LIN {X 0,Y 266.686,Z 225.636,A -85,B 0,C 180,E1 -19024.514,E2 -19024.514} C_VEL
LIN {X 0,Y 268.475,Z 213.294,A -85,B 0,C 180,E1 -19025.614,E2 -19025.614} C_VEL
LIN {X 0,Y 269.905,Z 200.622,A -85,B 0,C 180,E1 -19026.396,E2 -19026.396} C_VEL
LIN {X 0,Y 270.797,Z 187.768,A -85,B 0,C 180,E1 -19026.906,E2 -19026.906} C_VEL
LIN {X 0,Y 272.877,Z 131.801,A -85,B 0,C 180,E1 -19028.371,E2 -19028.371} C_VEL
LIN {X 0,Y 266.197,Z 116.896,A -85,B 0,C 180,E1 -19029.859,E2 -19029.859} C_VEL
LIN {X 0,Y 258.675,Z 102.48,A -85,B 0,C 180,E1 -19031.584,E2 -19031.584} C_VEL
LIN {X 0,Y 252.881,Z 93.623,A -85,B 0,C 180,E1 -19032.932,E2 -19032.932} C_VEL
LIN {X 0,Y 251.097,Z 90.671,A -85,B 0,C 180,E1 -19033.374,E2 -19033.374} C_VEL
LIN {X 0,Y 249.511,Z 88.379,A -85,B 0,C 180,E1 -19033.762,E2 -19033.762} C_VEL
LIN {X 0,Y 248.965,Z 86.456,A -85,B 0,C 180,E1 -19033.98,E2 -19033.98} C_VEL
LIN {X 0,Y 248.982,Z 86.472,A -85,B 0,C 180,E1 -19037.355,E2 -19037.355} C_VEL
LIN {X 0,Y 249.046,Z 86.459,A -85,B 0,C 180,E1 -19042.2,E2 -19042.2} C_VEL
LIN {X 0,Y 249.046,Z 86.459,A -85,B 0,C 180,E1 -19045.639,E2 -19045.639} C_VEL
LIN {X 0,Y 248.998,Z 86.463,A -85,B 0,C 180,E1 -19049.465,E2 -19049.465} C_VEL
LIN {X 0,Y 249.033,Z 86.454,A -85,B 0,C 180,E1 -19053.157,E2 -19053.157} C_VEL
LIN {X 0,Y 249.057,Z 86.45,A -85,B 0,C 180,E1 -19056.73,E2 -19056.73} C_VEL
LIN {X 0,Y 249.094,Z 86.457,A -85,B 0,C 180,E1 -19060.21,E2 -19060.21} C_VEL
LIN {X 0,Y 249.199,Z 86.435,A -85,B 0,C 180,E1 -19063.619,E2 -19063.619} C_VEL
LIN {X 0,Y 249.234,Z 86.424,A -85,B 0,C 180,E1 -19068.615,E2 -19068.615} C_VEL
LIN {X 0,Y 249.42,Z 86.413,A -85,B 0,C 180,E1 -19071.9,E2 -19071.9} C_VEL
LIN {X 0,Y 249.27,Z 86.425,A -85,B 0,C 180,E1 -19075.148,E2 -19075.148} C_VEL
LIN {X 0,Y 249.648,Z 86.375,A -85,B 0,C 180,E1 -19078.702,E2 -19078.702} C_VEL
LIN {X 0,Y 249.289,Z 86.416,A -85,B 0,C 180,E1 -19079.602,E2 -19079.602} C_VEL
LIN {X 0,Y 247.208,Z 86.686,A -85,B 0,C 180,E1 -19081.364,E2 -19081.364} C_VEL
LIN {X 0,Y 243.334,Z 87.169,A -85,B 0,C 180,E1 -19084.017,E2 -19084.017} C_VEL
LIN {X 0,Y 242.334,Z 87.282,A -85,B 0,C 180,E1 -19085.405,E2 -19085.405} C_VEL
LIN {X 0,Y 242.295,Z 87.285,A -85,B 0,C 180,E1 -19085.876,E2 -19085.876} C_VEL
LIN {X 0,Y 242.333,Z 87.296,A -85,B 0,C 180,E1 -19089.578,E2 -19089.578} C_VEL
LIN {X 0,Y 242.142,Z 87.321,A -85,B 0,C 180,E1 -19095.142,E2 -19095.142} C_VEL
LIN {X 0,Y 242.063,Z 87.326,A -85,B 0,C 180,E1 -19098.625,E2 -19098.625} C_VEL
LIN {X 0,Y 242.016,Z 87.324,A -85,B 0,C 180,E1 -19102.179,E2 -19102.179} C_VEL
LIN {X 0,Y 242.069,Z 87.326,A -85,B 0,C 180,E1 -19105.838,E2 -19105.838} C_VEL
LIN {X 0,Y 242.033,Z 87.335,A -85,B 0,C 180,E1 -19109.58,E2 -19109.58} C_VEL
LIN {X 0,Y 241.983,Z 87.341,A -85,B 0,C 180,E1 -19113.492,E2 -19113.492} C_VEL
LIN {X 0,Y 241.989,Z 87.313,A -85,B 0,C 180,E1 -19117.582,E2 -19117.582} C_VEL
LIN {X 0,Y 241.939,Z 87.346,A -85,B 0,C 180,E1 -19121.922,E2 -19121.922} C_VEL
LIN {X 0,Y 241.987,Z 87.448,A -85,B 0,C 180,E1 -19125.281,E2 -19125.281} C_VEL
LIN {X 0,Y 244.136,Z 95.03,A -85,B 0,C 180,E1 -19129.083,E2 -19129.083} C_VEL
LIN {X 0,Y 246.23,Z 102.697,A -85,B 0,C 180,E1 -19132.554,E2 -19132.554} C_VEL
LIN {X 0,Y 248.552,Z 107.076,A -85,B 0,C 180,E1 -19133.167,E2 -19133.167} C_VEL
LIN {X 0,Y 255.724,Z 121.344,A -85,B 0,C 180,E1 -19134.984,E2 -19134.984} C_VEL
LIN {X 0,Y 261.909,Z 135.149,A -85,B 0,C 180,E1 -19136.488,E2 -19136.488} C_VEL
LIN {X 0,Y 265.889,Z 160.561,A -85,B 0,C 180,E1 -19137.938,E2 -19137.938} C_VEL
LIN {X 0,Y 263.797,Z 212.777,A -85,B 0,C 180,E1 -19139.366,E2 -19139.366} C_VEL
LIN {X 0,Y 262.461,Z 226.52,A -85,B 0,C 180,E1 -19140.028,E2 -19140.028} C_VEL
LIN {X 0,Y 260.406,Z 239.381,A -85,B 0,C 180,E1 -19140.935,E2 -19140.935} C_VEL
LIN {X 0,Y 257.946,Z 251.892,A -85,B 0,C 180,E1 -19142.186,E2 -19142.186} C_VEL
LIN {X 0,Y 255.344,Z 263.061,A -85,B 0,C 180,E1 -19143.652,E2 -19143.652} C_VEL
LIN {X 0,Y 252.648,Z 273.135,A -85,B 0,C 180,E1 -19145.338,E2 -19145.338} C_VEL
LIN {X 0,Y 249.903,Z 282.245,A -85,B 0,C 180,E1 -19147.251,E2 -19147.251} C_VEL
LIN {X 0,Y 247.152,Z 291.145,A -85,B 0,C 180,E1 -19149.614,E2 -19149.614} C_VEL
LIN {X 0,Y 244.923,Z 298.327,A -85,B 0,C 180,E1 -19152.032,E2 -19152.032} C_VEL
LIN {X 0,Y 243.352,Z 303.192,A -85,B 0,C 180,E1 -19154.076,E2 -19154.076} C_VEL
LIN {X 0,Y 241.72,Z 307.936,A -85,B 0,C 180,E1 -19156.549,E2 -19156.549} C_VEL
LIN {X 0,Y 240.769,Z 311.589,A -85,B 0,C 180,E1 -19159.062,E2 -19159.062} C_VEL
LIN {X 0,Y 240.145,Z 314.246,A -85,B 0,C 180,E1 -19161.585,E2 -19161.585} C_VEL
LIN {X 0,Y 239.898,Z 315.513,A -85,B 0,C 180,E1 -19163.27,E2 -19163.27} C_VEL
LIN {X 0,Y 239.845,Z 316.4,A -85,B 0,C 180,E1 -19165.053,E2 -19165.053} C_VEL
LIN {X 0,Y 239.971,Z 316.852,A -85,B 0,C 180,E1 -19168.321,E2 -19168.321} C_VEL
LIN {X 0,Y 240.02,Z 316.509,A -85,B 0,C 180,E1 -19169.999,E2 -19169.999} C_VEL
LIN {X 0,Y 239.992,Z 315.759,A -85,B 0,C 180,E1 -19171.678,E2 -19171.678} C_VEL
LIN {X 0,Y 239.93,Z 314.556,A -85,B 0,C 180,E1 -19173.358,E2 -19173.358} C_VEL
LIN {X 0,Y 239.889,Z 311.975,A -85,B 0,C 180,E1 -19175.885,E2 -19175.885} C_VEL
LIN {X 0,Y 240.128,Z 308.368,A -85,B 0,C 180,E1 -19178.414,E2 -19178.414} C_VEL
LIN {X 0,Y 240.607,Z 303.629,A -85,B 0,C 180,E1 -19180.944,E2 -19180.944} C_VEL
LIN {X 0,Y 241.486,Z 297.624,A -85,B 0,C 180,E1 -19183.463,E2 -19183.463} C_VEL
LIN {X 0,Y 242.785,Z 290.138,A -85,B 0,C 180,E1 -19185.962,E2 -19185.962} C_VEL
LIN {X 0,Y 244.271,Z 282.197,A -85,B 0,C 180,E1 -19188.098,E2 -19188.098} C_VEL
LIN {X 0,Y 245.678,Z 273.231,A -85,B 0,C 180,E1 -19190.076,E2 -19190.076} C_VEL
LIN {X 0,Y 247.634,Z 262.952,A -85,B 0,C 180,E1 -19191.869,E2 -19191.869} C_VEL
LIN {X 0,Y 249.5,Z 251.528,A -85,B 0,C 180,E1 -19193.445,E2 -19193.445} C_VEL
LIN {X 0,Y 251.171,Z 239.655,A -85,B 0,C 180,E1 -19194.706,E2 -19194.706} C_VEL
LIN {X 0,Y 252.699,Z 226.572,A -85,B 0,C 180,E1 -19195.701,E2 -19195.701} C_VEL
LIN {X 0,Y 253.626,Z 213.267,A -85,B 0,C 180,E1 -19196.389,E2 -19196.389} C_VEL
LIN {X 0,Y 255.41,Z 156.007,A -85,B 0,C 180,E1 -19197.998,E2 -19197.998} C_VEL
LIN {X 0,Y 251.667,Z 125.16,A -85,B 0,C 180,E1 -19199.347,E2 -19199.347} C_VEL
LIN {X 0,Y 250.229,Z 115.793,A -85,B 0,C 180,E1 -19199.802,E2 -19199.802} C_VEL
LIN {X 0,Y 245.606,Z 103.483,A -85,B 0,C 180,E1 -19200.789,E2 -19200.789} C_VEL
LIN {X 0,Y 243.41,Z 93.051,A -85,B 0,C 180,E1 -19204.766,E2 -19204.766} C_VEL
LIN {X 0,Y 242.051,Z 87.339,A -85,B 0,C 180,E1 -19207.09,E2 -19207.09} C_VEL
LIN {X 0,Y 241.942,Z 87.348,A -85,B 0,C 180,E1 -19211.921,E2 -19211.921} C_VEL
LIN {X 0,Y 241.926,Z 87.349,A -85,B 0,C 180,E1 -19216.573,E2 -19216.573} C_VEL
LIN {X 0,Y 241.955,Z 87.332,A -85,B 0,C 180,E1 -19220.281,E2 -19220.281} C_VEL
LIN {X 0,Y 241.986,Z 87.339,A -85,B 0,C 180,E1 -19224.489,E2 -19224.489} C_VEL
LIN {X 0,Y 241.974,Z 87.343,A -85,B 0,C 180,E1 -19228.48,E2 -19228.48} C_VEL
LIN {X 0,Y 242.008,Z 87.336,A -85,B 0,C 180,E1 -19232.313,E2 -19232.313} C_VEL
LIN {X 0,Y 242.057,Z 87.332,A -85,B 0,C 180,E1 -19236.016,E2 -19236.016} C_VEL
LIN {X 0,Y 242.036,Z 87.324,A -85,B 0,C 180,E1 -19239.608,E2 -19239.608} C_VEL
LIN {X 0,Y 242.162,Z 87.319,A -85,B 0,C 180,E1 -19243.278,E2 -19243.278} C_VEL
LIN {X 0,Y 242.18,Z 87.305,A -85,B 0,C 180,E1 -19248.28,E2 -19248.28} C_VEL
LIN {X 0,Y 242.4,Z 87.289,A -85,B 0,C 180,E1 -19251.665,E2 -19251.665} C_VEL
LIN {X 0,Y 242.422,Z 87.285,A -85,B 0,C 180,E1 -19253.341,E2 -19253.341} C_VEL
LIN {X 0,Y 242.634,Z 87.258,A -85,B 0,C 180,E1 -19258.341,E2 -19258.341} C_VEL
LIN {X 0,Y 242.633,Z 87.261,A -85,B 0,C 180,E1 -19261.66,E2 -19261.66} C_VEL
LIN {X 0,Y 242.408,Z 87.284,A -85,B 0,C 180,E1 -19266.66,E2 -19266.66} C_VEL
LIN {X 0,Y 242.266,Z 87.304,A -85,B 0,C 180,E1 -19270.024,E2 -19270.024} C_VEL
LIN {X 0,Y 242.167,Z 87.312,A -85,B 0,C 180,E1 -19275.141,E2 -19275.141} C_VEL
LIN {X 0,Y 242.073,Z 87.327,A -85,B 0,C 180,E1 -19278.625,E2 -19278.625} C_VEL
LIN {X 0,Y 242.013,Z 87.329,A -85,B 0,C 180,E1 -19282.18,E2 -19282.18} C_VEL
LIN {X 0,Y 242.067,Z 87.33,A -85,B 0,C 180,E1 -19285.839,E2 -19285.839} C_VEL
LIN {X 0,Y 242.007,Z 87.338,A -85,B 0,C 180,E1 -19289.584,E2 -19289.584} C_VEL
LIN {X 0,Y 241.981,Z 87.342,A -85,B 0,C 180,E1 -19293.493,E2 -19293.493} C_VEL
LIN {X 0,Y 241.985,Z 87.34,A -85,B 0,C 180,E1 -19297.583,E2 -19297.583} C_VEL
LIN {X 0,Y 241.912,Z 87.349,A -85,B 0,C 180,E1 -19301.928,E2 -19301.928} C_VEL
LIN {X 0,Y 241.925,Z 87.351,A -85,B 0,C 180,E1 -19306.574,E2 -19306.574} C_VEL
LIN {X 0,Y 241.996,Z 87.34,A -85,B 0,C 180,E1 -19311.641,E2 -19311.641} C_VEL
LIN {X 0,Y 241.981,Z 87.343,A -85,B 0,C 180,E1 -19314.489,E2 -19314.489} C_VEL
LIN {X 0,Y 241.955,Z 87.346,A -85,B 0,C 180,E1 -19318.478,E2 -19318.478} C_VEL
LIN {X 0,Y 241.966,Z 87.336,A -85,B 0,C 180,E1 -19322.308,E2 -19322.308} C_VEL
LIN {X 0,Y 242.031,Z 87.516,A -85,B 0,C 180,E1 -19325.996,E2 -19325.996} C_VEL
LIN {X 0,Y 243.188,Z 90.492,A -85,B 0,C 180,E1 -19326.241,E2 -19326.241} C_VEL
LIN {X 0,Y 250.953,Z 106.159,A -85,B 0,C 180,E1 -19327.677,E2 -19327.677} C_VEL
LIN {X 0,Y 256.395,Z 121.2,A -85,B 0,C 180,E1 -19328.745,E2 -19328.745} C_VEL
LIN {X 0,Y 254.142,Z 192.259,A -85,B 0,C 180,E1 -19330.725,E2 -19330.725} C_VEL
LIN {X 0,Y 253.29,Z 205.938,A -85,B 0,C 180,E1 -19331.445,E2 -19331.445} C_VEL
LIN {X 0,Y 252.18,Z 218.733,A -85,B 0,C 180,E1 -19332.463,E2 -19332.463} C_VEL
LIN {X 0,Y 250.796,Z 230.411,A -85,B 0,C 180,E1 -19333.727,E2 -19333.727} C_VEL
LIN {X 0,Y 249.149,Z 241.669,A -85,B 0,C 180,E1 -19335.294,E2 -19335.294} C_VEL
LIN {X 0,Y 247.422,Z 251.831,A -85,B 0,C 180,E1 -19337.075,E2 -19337.075} C_VEL
LIN {X 0,Y 245.507,Z 261.778,A -85,B 0,C 180,E1 -19339.277,E2 -19339.277} C_VEL
LIN {X 0,Y 243.847,Z 270.522,A -85,B 0,C 180,E1 -19341.715,E2 -19341.715} C_VEL
LIN {X 0,Y 242.477,Z 277.536,A -85,B 0,C 180,E1 -19344.178,E2 -19344.178} C_VEL
LIN {X 0,Y 241.47,Z 283.133,A -85,B 0,C 180,E1 -19346.663,E2 -19346.663} C_VEL
LIN {X 0,Y 240.784,Z 287.545,A -85,B 0,C 180,E1 -19349.164,E2 -19349.164} C_VEL
LIN {X 0,Y 240.255,Z 290.905,A -85,B 0,C 180,E1 -19351.677,E2 -19351.677} C_VEL
LIN {X 0,Y 240.145,Z 292.572,A -85,B 0,C 180,E1 -19353.356,E2 -19353.356} C_VEL
LIN {X 0,Y 240.099,Z 294.188,A -85,B 0,C 180,E1 -19355.596,E2 -19355.596} C_VEL
LIN {X 0,Y 239.998,Z 295.194,A -85,B 0,C 180,E1 -19358.42,E2 -19358.42} C_VEL
LIN {X 0,Y 240.264,Z 294.941,A -85,B 0,C 180,E1 -19361.816,E2 -19361.816} C_VEL
LIN {X 0,Y 240.673,Z 294.231,A -85,B 0,C 180,E1 -19363.51,E2 -19363.51} C_VEL
LIN {X 0,Y 241.59,Z 292.169,A -85,B 0,C 180,E1 -19366.26,E2 -19366.26} C_VEL
LIN {X 0,Y 243.041,Z 288.332,A -85,B 0,C 180,E1 -19369.424,E2 -19369.424} C_VEL
LIN {X 0,Y 244.642,Z 284.067,A -85,B 0,C 180,E1 -19371.93,E2 -19371.93} C_VEL
LIN {X 0,Y 246.56,Z 278.599,A -85,B 0,C 180,E1 -19374.408,E2 -19374.408} C_VEL
LIN {X 0,Y 248.962,Z 271.704,A -85,B 0,C 180,E1 -19376.851,E2 -19376.851} C_VEL
LIN {X 0,Y 251.23,Z 264.642,A -85,B 0,C 180,E1 -19378.853,E2 -19378.853} C_VEL
LIN {X 0,Y 253.991,Z 254.913,A -85,B 0,C 180,E1 -19381.064,E2 -19381.064} C_VEL
LIN {X 0,Y 256.369,Z 245.433,A -85,B 0,C 180,E1 -19382.781,E2 -19382.781} C_VEL
LIN {X 0,Y 258.848,Z 234.847,A -85,B 0,C 180,E1 -19384.291,E2 -19384.291} C_VEL
LIN {X 0,Y 261.136,Z 223.08,A -85,B 0,C 180,E1 -19385.592,E2 -19385.592} C_VEL
LIN {X 0,Y 262.821,Z 210.853,A -85,B 0,C 180,E1 -19386.62,E2 -19386.62} C_VEL
LIN {X 0,Y 264.272,Z 197.71,A -85,B 0,C 180,E1 -19387.375,E2 -19387.375} C_VEL
LIN {X 0,Y 265.023,Z 184.983,A -85,B 0,C 180,E1 -19387.828,E2 -19387.828} C_VEL
LIN {X 0,Y 267.04,Z 133.98,A -85,B 0,C 180,E1 -19389.171,E2 -19389.171} C_VEL
LIN {X 0,Y 261.154,Z 120.766,A -85,B 0,C 180,E1 -19390.542,E2 -19390.542} C_VEL
LIN {X 0,Y 253.955,Z 106.895,A -85,B 0,C 180,E1 -19392.261,E2 -19392.261} C_VEL
LIN {X 0,Y 246.423,Z 95.208,A -85,B 0,C 180,E1 -19394.113,E2 -19394.113} C_VEL
LIN {X 0,Y 244.287,Z 91.787,A -85,B 0,C 180,E1 -19394.673,E2 -19394.673} C_VEL
LIN {X 0,Y 242.546,Z 89.488,A -85,B 0,C 180,E1 -19395.122,E2 -19395.122} C_VEL
LIN {X 0,Y 241.914,Z 87.332,A -85,B 0,C 180,E1 -19395.373,E2 -19395.373} C_VEL
LIN {X 0,Y 241.907,Z 87.348,A -85,B 0,C 180,E1 -19399.058,E2 -19399.058} C_VEL
LIN {X 0,Y 241.987,Z 87.34,A -85,B 0,C 180,E1 -19402.417,E2 -19402.417} C_VEL
LIN {X 0,Y 241.982,Z 87.343,A -85,B 0,C 180,E1 -19406.507,E2 -19406.507} C_VEL
LIN {X 0,Y 241.975,Z 87.344,A -85,B 0,C 180,E1 -19410.615,E2 -19410.615} C_VEL
LIN {X 0,Y 242.036,Z 87.334,A -85,B 0,C 180,E1 -19414.179,E2 -19414.179} C_VEL
LIN {X 0,Y 242.025,Z 87.329,A -85,B 0,C 180,E1 -19418.316,E2 -19418.316} C_VEL
LIN {X 0,Y 242.131,Z 87.312,A -85,B 0,C 180,E1 -19423.306,E2 -19423.306} C_VEL
LIN {X 0,Y 242.169,Z 87.302,A -85,B 0,C 180,E1 -19428.278,E2 -19428.278} C_VEL
LIN {X 0,Y 242.374,Z 87.293,A -85,B 0,C 180,E1 -19431.663,E2 -19431.663} C_VEL
LIN {X 0,Y 242.4,Z 87.274,A -85,B 0,C 180,E1 -19433.34,E2 -19433.34} C_VEL
LIN {X 0,Y 242.608,Z 87.252,A -85,B 0,C 180,E1 -19438.692,E2 -19438.692} C_VEL
LIN {X 0,Y 242.623,Z 87.257,A -85,B 0,C 180,E1 -19441.66,E2 -19441.66} C_VEL
LIN {X 0,Y 242.295,Z 87.285,A -85,B 0,C 180,E1 -19445.876,E2 -19445.876} C_VEL
LIN {X 0,Y 241.711,Z 87.366,A -85,B 0,C 180,E1 -19447.263,E2 -19447.263} C_VEL
LIN {X 0,Y 240.11,Z 87.574,A -85,B 0,C 180,E1 -19448.624,E2 -19448.624} C_VEL
LIN {X 0,Y 236.236,Z 88.046,A -85,B 0,C 180,E1 -19451.363,E2 -19451.363} C_VEL
LIN {X 0,Y 235.147,Z 88.18,A -85,B 0,C 180,E1 -19452.796,E2 -19452.796} C_VEL
LIN {X 0,Y 235.066,Z 88.192,A -85,B 0,C 180,E1 -19453.283,E2 -19453.283} C_VEL
LIN {X 0,Y 235.052,Z 88.189,A -85,B 0,C 180,E1 -19457.397,E2 -19457.397} C_VEL
LIN {X 0,Y 234.996,Z 88.198,A -85,B 0,C 180,E1 -19462.009,E2 -19462.009} C_VEL
LIN {X 0,Y 234.972,Z 88.205,A -85,B 0,C 180,E1 -19466.657,E2 -19466.657} C_VEL
LIN {X 0,Y 234.934,Z 88.212,A -85,B 0,C 180,E1 -19470.567,E2 -19470.567} C_VEL
LIN {X 0,Y 234.929,Z 88.201,A -85,B 0,C 180,E1 -19474.638,E2 -19474.638} C_VEL
LIN {X 0,Y 234.944,Z 88.212,A -85,B 0,C 180,E1 -19478.944,E2 -19478.944} C_VEL
LIN {X 0,Y 234.896,Z 88.281,A -85,B 0,C 180,E1 -19483.96,E2 -19483.96} C_VEL
LIN {X 0,Y 237.023,Z 95.585,A -85,B 0,C 180,E1 -19487.84,E2 -19487.84} C_VEL
LIN {X 0,Y 238.883,Z 102.23,A -85,B 0,C 180,E1 -19491.026,E2 -19491.026} C_VEL
LIN {X 0,Y 241.091,Z 106.391,A -85,B 0,C 180,E1 -19491.655,E2 -19491.655} C_VEL
LIN {X 0,Y 246.988,Z 117.484,A -85,B 0,C 180,E1 -19493.252,E2 -19493.252} C_VEL
LIN {X 0,Y 253.517,Z 131.294,A -85,B 0,C 180,E1 -19494.948,E2 -19494.948} C_VEL
LIN {X 0,Y 256.548,Z 138.573,A -85,B 0,C 180,E1 -19495.722,E2 -19495.722} C_VEL
LIN {X 0,Y 260.07,Z 161.624,A -85,B 0,C 180,E1 -19497.078,E2 -19497.078} C_VEL
LIN {X 0,Y 257.937,Z 212.151,A -85,B 0,C 180,E1 -19498.478,E2 -19498.478} C_VEL
LIN {X 0,Y 256.643,Z 225.227,A -85,B 0,C 180,E1 -19499.105,E2 -19499.105} C_VEL
LIN {X 0,Y 254.648,Z 237.853,A -85,B 0,C 180,E1 -19499.984,E2 -19499.984} C_VEL
LIN {X 0,Y 252.439,Z 249.089,A -85,B 0,C 180,E1 -19501.07,E2 -19501.07} C_VEL
LIN {X 0,Y 249.994,Z 259.425,A -85,B 0,C 180,E1 -19502.363,E2 -19502.363} C_VEL
LIN {X 0,Y 247.104,Z 270.114,A -85,B 0,C 180,E1 -19504.068,E2 -19504.068} C_VEL
LIN {X 0,Y 243.883,Z 280.635,A -85,B 0,C 180,E1 -19506.206,E2 -19506.206} C_VEL
LIN {X 0,Y 240.926,Z 289.756,A -85,B 0,C 180,E1 -19508.614,E2 -19508.614} C_VEL
LIN {X 0,Y 238.574,Z 297.128,A -85,B 0,C 180,E1 -19511.092,E2 -19511.092} C_VEL
LIN {X 0,Y 236.518,Z 303.063,A -85,B 0,C 180,E1 -19513.603,E2 -19513.603} C_VEL
LIN {X 0,Y 234.793,Z 307.765,A -85,B 0,C 180,E1 -19516.145,E2 -19516.145} C_VEL
LIN {X 0,Y 233.766,Z 311.379,A -85,B 0,C 180,E1 -19518.73,E2 -19518.73} C_VEL
LIN {X 0,Y 233.093,Z 314,A -85,B 0,C 180,E1 -19521.329,E2 -19521.329} C_VEL
LIN {X 0,Y 232.819,Z 315.249,A -85,B 0,C 180,E1 -19523.064,E2 -19523.064} C_VEL
LIN {X 0,Y 232.745,Z 316.188,A -85,B 0,C 180,E1 -19525.185,E2 -19525.185} C_VEL
LIN {X 0,Y 232.898,Z 316.524,A -85,B 0,C 180,E1 -19528.27,E2 -19528.27} C_VEL
LIN {X 0,Y 232.947,Z 316.165,A -85,B 0,C 180,E1 -19529.999,E2 -19529.999} C_VEL
LIN {X 0,Y 232.92,Z 315.383,A -85,B 0,C 180,E1 -19531.729,E2 -19531.729} C_VEL
LIN {X 0,Y 232.801,Z 312.753,A -85,B 0,C 180,E1 -19534.974,E2 -19534.974} C_VEL
LIN {X 0,Y 232.966,Z 309.225,A -85,B 0,C 180,E1 -19537.802,E2 -19537.802} C_VEL
LIN {X 0,Y 233.391,Z 304.837,A -85,B 0,C 180,E1 -19540.409,E2 -19540.409} C_VEL
LIN {X 0,Y 234.155,Z 299.239,A -85,B 0,C 180,E1 -19543.009,E2 -19543.009} C_VEL
LIN {X 0,Y 235.443,Z 292.254,A -85,B 0,C 180,E1 -19545.583,E2 -19545.583} C_VEL
LIN {X 0,Y 237.033,Z 284.158,A -85,B 0,C 180,E1 -19547.957,E2 -19547.957} C_VEL
LIN {X 0,Y 238.594,Z 274.467,A -85,B 0,C 180,E1 -19550.249,E2 -19550.249} C_VEL
LIN {X 0,Y 240.547,Z 264.596,A -85,B 0,C 180,E1 -19552.096,E2 -19552.096} C_VEL
LIN {X 0,Y 242.469,Z 253.719,A -85,B 0,C 180,E1 -19553.713,E2 -19553.713} C_VEL
LIN {X 0,Y 244.299,Z 241.486,A -85,B 0,C 180,E1 -19555.108,E2 -19555.108} C_VEL
LIN {X 0,Y 245.939,Z 228.696,A -85,B 0,C 180,E1 -19556.176,E2 -19556.176} C_VEL
LIN {X 0,Y 246.944,Z 215.883,A -85,B 0,C 180,E1 -19556.916,E2 -19556.916} C_VEL
LIN {X 0,Y 247.636,Z 199.657,A -85,B 0,C 180,E1 -19557.457,E2 -19557.457} C_VEL
LIN {X 0,Y 248.905,Z 156.447,A -85,B 0,C 180,E1 -19558.673,E2 -19558.673} C_VEL
LIN {X 0,Y 245.449,Z 127.202,A -85,B 0,C 180,E1 -19559.991,E2 -19559.991} C_VEL
LIN {X 0,Y 244.025,Z 118.013,A -85,B 0,C 180,E1 -19560.456,E2 -19560.456} C_VEL
LIN {X 0,Y 239.176,Z 105.676,A -85,B 0,C 180,E1 -19561.463,E2 -19561.463} C_VEL
LIN {X 0,Y 238.303,Z 103.126,A -85,B 0,C 180,E1 -19561.713,E2 -19561.713} C_VEL
LIN {X 0,Y 236.632,Z 95.125,A -85,B 0,C 180,E1 -19564.87,E2 -19564.87} C_VEL
LIN {X 0,Y 234.976,Z 88.221,A -85,B 0,C 180,E1 -19567.817,E2 -19567.817} C_VEL
LIN {X 0,Y 234.891,Z 88.226,A -85,B 0,C 180,E1 -19571.582,E2 -19571.582} C_VEL
LIN {X 0,Y 234.887,Z 88.227,A -85,B 0,C 180,E1 -19575.897,E2 -19575.897} C_VEL
LIN {X 0,Y 234.881,Z 88.225,A -85,B 0,C 180,E1 -19578.832,E2 -19578.832} C_VEL
LIN {X 0,Y 234.916,Z 88.203,A -85,B 0,C 180,E1 -19581.079,E2 -19581.079} C_VEL
LIN {X 0,Y 234.929,Z 88.222,A -85,B 0,C 180,E1 -19585.362,E2 -19585.362} C_VEL
LIN {X 0,Y 234.931,Z 88.221,A -85,B 0,C 180,E1 -19589.432,E2 -19589.432} C_VEL
LIN {X 0,Y 234.993,Z 88.206,A -85,B 0,C 180,E1 -19593.794,E2 -19593.794} C_VEL
LIN {X 0,Y 235.011,Z 88.201,A -85,B 0,C 180,E1 -19598.97,E2 -19598.97} C_VEL
LIN {X 0,Y 235.096,Z 88.2,A -85,B 0,C 180,E1 -19603.059,E2 -19603.059} C_VEL
LIN {X 0,Y 235.114,Z 88.183,A -85,B 0,C 180,E1 -19607.922,E2 -19607.922} C_VEL
LIN {X 0,Y 235.331,Z 88.17,A -85,B 0,C 180,E1 -19611.413,E2 -19611.413} C_VEL
LIN {X 0,Y 235.373,Z 88.163,A -85,B 0,C 180,E1 -19613.141,E2 -19613.141} C_VEL
LIN {X 0,Y 235.593,Z 88.134,A -85,B 0,C 180,E1 -19618.291,E2 -19618.291} C_VEL
LIN {X 0,Y 235.593,Z 88.138,A -85,B 0,C 180,E1 -19621.71,E2 -19621.71} C_VEL
LIN {X 0,Y 235.359,Z 88.161,A -85,B 0,C 180,E1 -19626.86,E2 -19626.86} C_VEL
LIN {X 0,Y 235.212,Z 88.181,A -85,B 0,C 180,E1 -19630.328,E2 -19630.328} C_VEL
LIN {X 0,Y 235.114,Z 88.193,A -85,B 0,C 180,E1 -19635.607,E2 -19635.607} C_VEL
LIN {X 0,Y 235.009,Z 88.207,A -85,B 0,C 180,E1 -19639.206,E2 -19639.206} C_VEL
LIN {X 0,Y 234.961,Z 88.208,A -85,B 0,C 180,E1 -19642.883,E2 -19642.883} C_VEL
LIN {X 0,Y 234.968,Z 88.214,A -85,B 0,C 180,E1 -19646.658,E2 -19646.658} C_VEL
LIN {X 0,Y 234.923,Z 88.22,A -85,B 0,C 180,E1 -19650.57,E2 -19650.57} C_VEL
LIN {X 0,Y 234.927,Z 88.221,A -85,B 0,C 180,E1 -19654.639,E2 -19654.639} C_VEL
LIN {X 0,Y 234.912,Z 88.224,A -85,B 0,C 180,E1 -19658.936,E2 -19658.936} C_VEL
LIN {X 0,Y 234.865,Z 88.229,A -85,B 0,C 180,E1 -19663.492,E2 -19663.492} C_VEL
LIN {X 0,Y 234.878,Z 88.229,A -85,B 0,C 180,E1 -19666.513,E2 -19666.513} C_VEL
LIN {X 0,Y 234.919,Z 88.222,A -85,B 0,C 180,E1 -19671.079,E2 -19671.079} C_VEL
LIN {X 0,Y 234.927,Z 88.22,A -85,B 0,C 180,E1 -19675.362,E2 -19675.362} C_VEL
LIN {X 0,Y 234.901,Z 88.222,A -85,B 0,C 180,E1 -19679.428,E2 -19679.428} C_VEL
LIN {X 0,Y 234.966,Z 88.216,A -85,B 0,C 180,E1 -19684.394,E2 -19684.394} C_VEL
LIN {X 0,Y 234.994,Z 88.214,A -85,B 0,C 180,E1 -19685.069,E2 -19685.069} C_VEL
LIN {X 0,Y 236.009,Z 91.114,A -85,B 0,C 180,E1 -19685.329,E2 -19685.329} C_VEL
LIN {X 0,Y 244.946,Z 108.846,A -85,B 0,C 180,E1 -19687.056,E2 -19687.056} C_VEL
LIN {X 0,Y 249.986,Z 122.737,A -85,B 0,C 180,E1 -19688.088,E2 -19688.088} C_VEL
LIN {X 0,Y 247.68,Z 191.908,A -85,B 0,C 180,E1 -19690.047,E2 -19690.047} C_VEL
LIN {X 0,Y 246.882,Z 204.939,A -85,B 0,C 180,E1 -19690.729,E2 -19690.729} C_VEL
LIN {X 0,Y 245.681,Z 218.154,A -85,B 0,C 180,E1 -19691.768,E2 -19691.768} C_VEL
LIN {X 0,Y 244.278,Z 230.044,A -85,B 0,C 180,E1 -19693.065,E2 -19693.065} C_VEL
LIN {X 0,Y 242.541,Z 241.43,A -85,B 0,C 180,E1 -19694.669,E2 -19694.669} C_VEL
LIN {X 0,Y 240.757,Z 251.696,A -85,B 0,C 180,E1 -19696.496,E2 -19696.496} C_VEL
LIN {X 0,Y 238.931,Z 260.935,A -85,B 0,C 180,E1 -19698.549,E2 -19698.549} C_VEL
LIN {X 0,Y 237.116,Z 269.879,A -85,B 0,C 180,E1 -19701.048,E2 -19701.048} C_VEL
LIN {X 0,Y 235.671,Z 277.088,A -85,B 0,C 180,E1 -19703.58,E2 -19703.58} C_VEL
LIN {X 0,Y 234.691,Z 281.968,A -85,B 0,C 180,E1 -19705.707,E2 -19705.707} C_VEL
LIN {X 0,Y 233.917,Z 286.706,A -85,B 0,C 180,E1 -19708.279,E2 -19708.279} C_VEL
LIN {X 0,Y 233.284,Z 290.357,A -85,B 0,C 180,E1 -19710.864,E2 -19710.864} C_VEL
LIN {X 0,Y 233.051,Z 292.996,A -85,B 0,C 180,E1 -19713.458,E2 -19713.458} C_VEL
LIN {X 0,Y 233.032,Z 294.479,A -85,B 0,C 180,E1 -19715.582,E2 -19715.582} C_VEL
LIN {X 0,Y 232.906,Z 295.529,A -85,B 0,C 180,E1 -19718.678,E2 -19718.678} C_VEL
LIN {X 0,Y 233.237,Z 295.231,A -85,B 0,C 180,E1 -19722.177,E2 -19722.177} C_VEL
LIN {X 0,Y 233.704,Z 294.485,A -85,B 0,C 180,E1 -19723.921,E2 -19723.921} C_VEL
LIN {X 0,Y 234.613,Z 292.567,A -85,B 0,C 180,E1 -19726.545,E2 -19726.545} C_VEL
LIN {X 0,Y 235.78,Z 289.692,A -85,B 0,C 180,E1 -19729.141,E2 -19729.141} C_VEL
LIN {X 0,Y 237.351,Z 285.752,A -85,B 0,C 180,E1 -19731.724,E2 -19731.724} C_VEL
LIN {X 0,Y 239.484,Z 280.052,A -85,B 0,C 180,E1 -19734.529,E2 -19734.529} C_VEL
LIN {X 0,Y 242.11,Z 272.914,A -85,B 0,C 180,E1 -19737.207,E2 -19737.207} C_VEL
LIN {X 0,Y 244.946,Z 264.531,A -85,B 0,C 180,E1 -19739.666,E2 -19739.666} C_VEL
LIN {X 0,Y 247.715,Z 255.097,A -85,B 0,C 180,E1 -19741.84,E2 -19741.84} C_VEL
LIN {X 0,Y 250.042,Z 246.27,A -85,B 0,C 180,E1 -19743.478,E2 -19743.478} C_VEL
LIN {X 0,Y 252.607,Z 235.795,A -85,B 0,C 180,E1 -19745.018,E2 -19745.018} C_VEL
LIN {X 0,Y 254.989,Z 224.255,A -85,B 0,C 180,E1 -19746.341,E2 -19746.341} C_VEL
LIN {X 0,Y 256.643,Z 212.885,A -85,B 0,C 180,E1 -19747.352,E2 -19747.352} C_VEL
LIN {X 0,Y 258.232,Z 199.432,A -85,B 0,C 180,E1 -19748.172,E2 -19748.172} C_VEL
LIN {X 0,Y 259.127,Z 186.818,A -85,B 0,C 180,E1 -19748.653,E2 -19748.653} C_VEL
LIN {X 0,Y 261.218,Z 136.002,A -85,B 0,C 180,E1 -19750.019,E2 -19750.019} C_VEL
LIN {X 0,Y 255.346,Z 123.018,A -85,B 0,C 180,E1 -19751.447,E2 -19751.447} C_VEL
LIN {X 0,Y 249.181,Z 111.171,A -85,B 0,C 180,E1 -19752.987,E2 -19752.987} C_VEL
LIN {X 0,Y 241.952,Z 99.851,A -85,B 0,C 180,E1 -19754.844,E2 -19754.844} C_VEL
LIN {X 0,Y 239.574,Z 96.295,A -85,B 0,C 180,E1 -19755.484,E2 -19755.484} C_VEL
LIN {X 0,Y 237.264,Z 92.721,A -85,B 0,C 180,E1 -19756.131,E2 -19756.131} C_VEL
LIN {X 0,Y 235.438,Z 90.284,A -85,B 0,C 180,E1 -19756.64,E2 -19756.64} C_VEL
LIN {X 0,Y 234.873,Z 88.227,A -85,B 0,C 180,E1 -19756.902,E2 -19756.902} C_VEL
LIN {X 0,Y 234.921,Z 88.217,A -85,B 0,C 180,E1 -19761.078,E2 -19761.078} C_VEL
LIN {X 0,Y 234.926,Z 88.215,A -85,B 0,C 180,E1 -19765.36,E2 -19765.36} C_VEL
LIN {X 0,Y 234.898,Z 88.219,A -85,B 0,C 180,E1 -19769.427,E2 -19769.427} C_VEL
LIN {X 0,Y 234.971,Z 88.21,A -85,B 0,C 180,E1 -19773.807,E2 -19773.807} C_VEL
LIN {X 0,Y 234.994,Z 88.209,A -85,B 0,C 180,E1 -19778.968,E2 -19778.968} C_VEL
LIN {X 0,Y 235.067,Z 88.19,A -85,B 0,C 180,E1 -19783.085,E2 -19783.085} C_VEL
LIN {X 0,Y 235.101,Z 88.182,A -85,B 0,C 180,E1 -19787.921,E2 -19787.921} C_VEL
LIN {X 0,Y 235.314,Z 88.173,A -85,B 0,C 180,E1 -19791.411,E2 -19791.411} C_VEL
LIN {X 0,Y 235.351,Z 88.152,A -85,B 0,C 180,E1 -19793.139,E2 -19793.139} C_VEL
LIN {X 0,Y 235.581,Z 88.131,A -85,B 0,C 180,E1 -19798.29,E2 -19798.29} C_VEL
LIN {X 0,Y 235.582,Z 88.134,A -85,B 0,C 180,E1 -19801.709,E2 -19801.709} C_VEL
LIN {X 0,Y 235.356,Z 88.153,A -85,B 0,C 180,E1 -19806.86,E2 -19806.86} C_VEL
LIN {X 0,Y 235.215,Z 88.176,A -85,B 0,C 180,E1 -19810.327,E2 -19810.327} C_VEL
LIN {X 0,Y 235.066,Z 88.192,A -85,B 0,C 180,E1 -19813.283,E2 -19813.283} C_VEL
LIN {X 0,Y 234.402,Z 88.288,A -85,B 0,C 180,E1 -19814.713,E2 -19814.713} C_VEL
LIN {X 0,Y 231.497,Z 88.655,A -85,B 0,C 180,E1 -19817.044,E2 -19817.044} C_VEL
LIN {X 0,Y 229.033,Z 88.955,A -85,B 0,C 180,E1 -19818.946,E2 -19818.946} C_VEL
LIN {X 0,Y 227.997,Z 89.083,A -85,B 0,C 180,E1 -19820.423,E2 -19820.423} C_VEL
LIN {X 0,Y 227.924,Z 89.082,A -85,B 0,C 180,E1 -19820.924,E2 -19820.924} C_VEL
LIN {X 0,Y 227.932,Z 89.088,A -85,B 0,C 180,E1 -19825.574,E2 -19825.574} C_VEL
LIN {X 0,Y 227.911,Z 89.088,A -85,B 0,C 180,E1 -19830.295,E2 -19830.295} C_VEL
LIN {X 0,Y 227.879,Z 89.095,A -85,B 0,C 180,E1 -19833.72,E2 -19833.72} C_VEL
LIN {X 0,Y 227.846,Z 89.079,A -85,B 0,C 180,E1 -19838.09,E2 -19838.09} C_VEL
LIN {X 0,Y 227.824,Z 89.217,A -85,B 0,C 180,E1 -19842.576,E2 -19842.576} C_VEL
LIN {X 0,Y 230.218,Z 97.3,A -85,B 0,C 180,E1 -19847.11,E2 -19847.11} C_VEL
LIN {X 0,Y 231.416,Z 101.635,A -85,B 0,C 180,E1 -19849.325,E2 -19849.325} C_VEL
LIN {X 0,Y 234.033,Z 106.264,A -85,B 0,C 180,E1 -19850.121,E2 -19850.121} C_VEL
LIN {X 0,Y 240.008,Z 117.265,A -85,B 0,C 180,E1 -19851.853,E2 -19851.853} C_VEL
LIN {X 0,Y 245.83,Z 129.069,A -85,B 0,C 180,E1 -19853.46,E2 -19853.46} C_VEL
LIN {X 0,Y 251.034,Z 140.891,A -85,B 0,C 180,E1 -19854.849,E2 -19854.849} C_VEL
LIN {X 0,Y 254.305,Z 162.569,A -85,B 0,C 180,E1 -19856.173,E2 -19856.173} C_VEL
LIN {X 0,Y 252.08,Z 212.308,A -85,B 0,C 180,E1 -19857.581,E2 -19857.581} C_VEL
LIN {X 0,Y 250.623,Z 226.204,A -85,B 0,C 180,E1 -19858.278,E2 -19858.278} C_VEL
LIN {X 0,Y 248.55,Z 238.451,A -85,B 0,C 180,E1 -19859.169,E2 -19859.169} C_VEL
LIN {X 0,Y 245.886,Z 251.024,A -85,B 0,C 180,E1 -19860.458,E2 -19860.458} C_VEL
LIN {X 0,Y 243.046,Z 262.235,A -85,B 0,C 180,E1 -19861.972,E2 -19861.972} C_VEL
LIN {X 0,Y 240.155,Z 272.351,A -85,B 0,C 180,E1 -19863.728,E2 -19863.728} C_VEL
LIN {X 0,Y 236.86,Z 282.298,A -85,B 0,C 180,E1 -19865.921,E2 -19865.921} C_VEL
LIN {X 0,Y 233.86,Z 291.081,A -85,B 0,C 180,E1 -19868.399,E2 -19868.399} C_VEL
LIN {X 0,Y 231.451,Z 298.127,A -85,B 0,C 180,E1 -19870.948,E2 -19870.948} C_VEL
LIN {X 0,Y 229.04,Z 304.596,A -85,B 0,C 180,E1 -19873.968,E2 -19873.968} C_VEL
LIN {X 0,Y 227.447,Z 308.883,A -85,B 0,C 180,E1 -19876.6,E2 -19876.6} C_VEL
LIN {X 0,Y 226.496,Z 312.127,A -85,B 0,C 180,E1 -19879.27,E2 -19879.27} C_VEL
LIN {X 0,Y 225.765,Z 314.984,A -85,B 0,C 180,E1 -19882.846,E2 -19882.846} C_VEL
LIN {X 0,Y 225.674,Z 316.178,A -85,B 0,C 180,E1 -19886.428,E2 -19886.428} C_VEL
LIN {X 0,Y 225.802,Z 316.195,A -85,B 0,C 180,E1 -19888.216,E2 -19888.216} C_VEL
LIN {X 0,Y 225.877,Z 315.819,A -85,B 0,C 180,E1 -19889.999,E2 -19889.999} C_VEL
LIN {X 0,Y 225.826,Z 315.003,A -85,B 0,C 180,E1 -19891.783,E2 -19891.783} C_VEL
LIN {X 0,Y 225.726,Z 312.555,A -85,B 0,C 180,E1 -19894.916,E2 -19894.916} C_VEL
LIN {X 0,Y 225.89,Z 308.769,A -85,B 0,C 180,E1 -19898.048,E2 -19898.048} C_VEL
LIN {X 0,Y 226.347,Z 304.34,A -85,B 0,C 180,E1 -19900.736,E2 -19900.736} C_VEL
LIN {X 0,Y 227.181,Z 298.698,A -85,B 0,C 180,E1 -19903.415,E2 -19903.415} C_VEL
LIN {X 0,Y 228.533,Z 291.651,A -85,B 0,C 180,E1 -19906.067,E2 -19906.067} C_VEL
LIN {X 0,Y 230.071,Z 284.33,A -85,B 0,C 180,E1 -19908.283,E2 -19908.283} C_VEL
LIN {X 0,Y 231.528,Z 275.698,A -85,B 0,C 180,E1 -19910.431,E2 -19910.431} C_VEL
LIN {X 0,Y 233.711,Z 264.952,A -85,B 0,C 180,E1 -19912.545,E2 -19912.545} C_VEL
LIN {X 0,Y 235.686,Z 254.266,A -85,B 0,C 180,E1 -19914.205,E2 -19914.205} C_VEL
LIN {X 0,Y 237.569,Z 242.309,A -85,B 0,C 180,E1 -19915.635,E2 -19915.635} C_VEL
LIN {X 0,Y 239.245,Z 229.867,A -85,B 0,C 180,E1 -19916.731,E2 -19916.731} C_VEL
LIN {X 0,Y 240.391,Z 216.995,A -85,B 0,C 180,E1 -19917.534,E2 -19917.534} C_VEL
LIN {X 0,Y 241.071,Z 203.419,A -85,B 0,C 180,E1 -19918.035,E2 -19918.035} C_VEL
LIN {X 0,Y 242.463,Z 156.9,A -85,B 0,C 180,E1 -19919.38,E2 -19919.38} C_VEL
LIN {X 0,Y 239.228,Z 129.017,A -85,B 0,C 180,E1 -19920.68,E2 -19920.68} C_VEL
LIN {X 0,Y 237.852,Z 120.034,A -85,B 0,C 180,E1 -19921.151,E2 -19921.151} C_VEL
LIN {X 0,Y 232.052,Z 105.517,A -85,B 0,C 180,E1 -19922.41,E2 -19922.41} C_VEL
LIN {X 0,Y 231.023,Z 102.805,A -85,B 0,C 180,E1 -19922.683,E2 -19922.683} C_VEL
LIN {X 0,Y 229.254,Z 94.549,A -85,B 0,C 180,E1 -19926.097,E2 -19926.097} C_VEL
LIN {X 0,Y 227.916,Z 89.097,A -85,B 0,C 180,E1 -19928.543,E2 -19928.543} C_VEL
LIN {X 0,Y 227.812,Z 89.108,A -85,B 0,C 180,E1 -19932.742,E2 -19932.742} C_VEL
LIN {X 0,Y 227.806,Z 89.109,A -85,B 0,C 180,E1 -19937.257,E2 -19937.257} C_VEL
LIN {X 0,Y 227.842,Z 89.084,A -85,B 0,C 180,E1 -19941.909,E2 -19941.909} C_VEL
LIN {X 0,Y 227.878,Z 89.097,A -85,B 0,C 180,E1 -19946.377,E2 -19946.377} C_VEL
LIN {X 0,Y 227.918,Z 89.094,A -85,B 0,C 180,E1 -19950.438,E2 -19950.438} C_VEL
LIN {X 0,Y 227.928,Z 89.087,A -85,B 0,C 180,E1 -19954.426,E2 -19954.426} C_VEL
LIN {X 0,Y 227.961,Z 89.085,A -85,B 0,C 180,E1 -19958.287,E2 -19958.287} C_VEL
LIN {X 0,Y 228.034,Z 89.081,A -85,B 0,C 180,E1 -19962.826,E2 -19962.826} C_VEL
LIN {X 0,Y 228.072,Z 89.059,A -85,B 0,C 180,E1 -19967.543,E2 -19967.543} C_VEL
LIN {X 0,Y 228.267,Z 89.05,A -85,B 0,C 180,E1 -19971.145,E2 -19971.145} C_VEL
LIN {X 0,Y 228.323,Z 89.042,A -85,B 0,C 180,E1 -19972.928,E2 -19972.928} C_VEL
LIN {X 0,Y 228.552,Z 89.01,A -85,B 0,C 180,E1 -19978.238,E2 -19978.238} C_VEL
LIN {X 0,Y 228.551,Z 89.015,A -85,B 0,C 180,E1 -19981.763,E2 -19981.763} C_VEL
LIN {X 0,Y 228.311,Z 89.039,A -85,B 0,C 180,E1 -19987.073,E2 -19987.073} C_VEL
LIN {X 0,Y 228.142,Z 89.061,A -85,B 0,C 180,E1 -19990.652,E2 -19990.652} C_VEL
LIN {X 0,Y 228.057,Z 89.067,A -85,B 0,C 180,E1 -19994.273,E2 -19994.273} C_VEL
LIN {X 0,Y 228.003,Z 89.081,A -85,B 0,C 180,E1 -19997.954,E2 -19997.954} C_VEL
LIN {X 0,Y 227.93,Z 89.082,A -85,B 0,C 180,E1 -20002.33,E2 -20002.33} C_VEL
LIN {X 0,Y 227.942,Z 89.089,A -85,B 0,C 180,E1 -20006.603,E2 -20006.603} C_VEL
LIN {X 0,Y 227.897,Z 89.095,A -85,B 0,C 180,E1 -20010.292,E2 -20010.292} C_VEL
LIN {X 0,Y 227.877,Z 89.098,A -85,B 0,C 180,E1 -20013.721,E2 -20013.721} C_VEL
LIN {X 0,Y 227.843,Z 89.102,A -85,B 0,C 180,E1 -20018.092,E2 -20018.092} C_VEL
LIN {X 0,Y 227.792,Z 89.112,A -85,B 0,C 180,E1 -20022.748,E2 -20022.748} C_VEL
LIN {X 0,Y 227.804,Z 89.106,A -85,B 0,C 180,E1 -20027.257,E2 -20027.257} C_VEL
LIN {X 0,Y 227.841,Z 89.104,A -85,B 0,C 180,E1 -20031.909,E2 -20031.909} C_VEL
LIN {X 0,Y 227.88,Z 89.096,A -85,B 0,C 180,E1 -20036.378,E2 -20036.378} C_VEL
LIN {X 0,Y 227.878,Z 89.086,A -85,B 0,C 180,E1 -20040.432,E2 -20040.432} C_VEL
LIN {X 0,Y 227.931,Z 89.093,A -85,B 0,C 180,E1 -20044.104,E2 -20044.104} C_VEL
LIN {X 0,Y 228.928,Z 91.953,A -85,B 0,C 180,E1 -20044.373,E2 -20044.373} C_VEL
LIN {X 0,Y 236.223,Z 105.971,A -85,B 0,C 180,E1 -20045.863,E2 -20045.863} C_VEL
LIN {X 0,Y 239.987,Z 114.135,A -85,B 0,C 180,E1 -20046.62,E2 -20046.62} C_VEL
LIN {X 0,Y 243.607,Z 124.372,A -85,B 0,C 180,E1 -20047.399,E2 -20047.399} C_VEL
LIN {X 0,Y 241.215,Z 192.535,A -85,B 0,C 180,E1 -20049.377,E2 -20049.377} C_VEL
LIN {X 0,Y 240.303,Z 206.212,A -85,B 0,C 180,E1 -20050.124,E2 -20050.124} C_VEL
LIN {X 0,Y 239.141,Z 218.61,A -85,B 0,C 180,E1 -20051.139,E2 -20051.139} C_VEL
LIN {X 0,Y 237.788,Z 229.678,A -85,B 0,C 180,E1 -20052.366,E2 -20052.366} C_VEL
LIN {X 0,Y 235.981,Z 241.188,A -85,B 0,C 180,E1 -20054.01,E2 -20054.01} C_VEL
LIN {X 0,Y 234.09,Z 251.554,A -85,B 0,C 180,E1 -20055.882,E2 -20055.882} C_VEL
LIN {X 0,Y 232.355,Z 260.038,A -85,B 0,C 180,E1 -20057.777,E2 -20057.777} C_VEL
LIN {X 0,Y 230.748,Z 267.856,A -85,B 0,C 180,E1 -20059.914,E2 -20059.914} C_VEL
LIN {X 0,Y 229.061,Z 275.507,A -85,B 0,C 180,E1 -20062.508,E2 -20062.508} C_VEL
LIN {X 0,Y 227.638,Z 282.541,A -85,B 0,C 180,E1 -20065.574,E2 -20065.574} C_VEL
LIN {X 0,Y 226.826,Z 287.227,A -85,B 0,C 180,E1 -20068.225,E2 -20068.225} C_VEL
LIN {X 0,Y 226.192,Z 290.827,A -85,B 0,C 180,E1 -20070.891,E2 -20070.891} C_VEL
LIN {X 0,Y 225.963,Z 293.418,A -85,B 0,C 180,E1 -20073.567,E2 -20073.567} C_VEL
LIN {X 0,Y 225.96,Z 294.761,A -85,B 0,C 180,E1 -20075.556,E2 -20075.556} C_VEL
LIN {X 0,Y 225.836,Z 295.863,A -85,B 0,C 180,E1 -20078.952,E2 -20078.952} C_VEL
LIN {X 0,Y 226.224,Z 295.52,A -85,B 0,C 180,E1 -20082.561,E2 -20082.561} C_VEL
LIN {X 0,Y 226.734,Z 294.73,A -85,B 0,C 180,E1 -20084.358,E2 -20084.358} C_VEL
LIN {X 0,Y 227.604,Z 292.988,A -85,B 0,C 180,E1 -20086.816,E2 -20086.816} C_VEL
LIN {X 0,Y 228.99,Z 289.857,A -85,B 0,C 180,E1 -20089.732,E2 -20089.732} C_VEL
LIN {X 0,Y 230.647,Z 285.864,A -85,B 0,C 180,E1 -20092.389,E2 -20092.389} C_VEL
LIN {X 0,Y 232.739,Z 280.588,A -85,B 0,C 180,E1 -20095.053,E2 -20095.053} C_VEL
LIN {X 0,Y 235.245,Z 274.123,A -85,B 0,C 180,E1 -20097.586,E2 -20097.586} C_VEL
LIN {X 0,Y 238.153,Z 265.935,A -85,B 0,C 180,E1 -20100.112,E2 -20100.112} C_VEL
LIN {X 0,Y 240.883,Z 257.398,A -85,B 0,C 180,E1 -20102.208,E2 -20102.208} C_VEL
LIN {X 0,Y 243.453,Z 248.291,A -85,B 0,C 180,E1 -20104.009,E2 -20104.009} C_VEL
LIN {X 0,Y 246.087,Z 238.186,A -85,B 0,C 180,E1 -20105.584,E2 -20105.584} C_VEL
LIN {X 0,Y 248.508,Z 227.148,A -85,B 0,C 180,E1 -20106.94,E2 -20106.94} C_VEL
LIN {X 0,Y 250.535,Z 214.868,A -85,B 0,C 180,E1 -20108.108,E2 -20108.108} C_VEL
LIN {X 0,Y 252.182,Z 201.993,A -85,B 0,C 180,E1 -20108.961,E2 -20108.961} C_VEL
LIN {X 0,Y 253.262,Z 188.191,A -85,B 0,C 180,E1 -20109.533,E2 -20109.533} C_VEL
LIN {X 0,Y 255.381,Z 138.011,A -85,B 0,C 180,E1 -20110.919,E2 -20110.919} C_VEL
LIN {X 0,Y 249.121,Z 124.271,A -85,B 0,C 180,E1 -20112.521,E2 -20112.521} C_VEL
LIN {X 0,Y 244.289,Z 115.147,A -85,B 0,C 180,E1 -20113.785,E2 -20113.785} C_VEL
LIN {X 0,Y 237.538,Z 104.451,A -85,B 0,C 180,E1 -20115.6,E2 -20115.6} C_VEL
LIN {X 0,Y 233.009,Z 97.683,A -85,B 0,C 180,E1 -20116.893,E2 -20116.893} C_VEL
LIN {X 0,Y 230.862,Z 94.251,A -85,B 0,C 180,E1 -20117.543,E2 -20117.543} C_VEL
LIN {X 0,Y 228.617,Z 91.624,A -85,B 0,C 180,E1 -20118.202,E2 -20118.202} C_VEL
LIN {X 0,Y 227.834,Z 89.099,A -85,B 0,C 180,E1 -20118.563,E2 -20118.563} C_VEL
LIN {X 0,Y 227.883,Z 89.099,A -85,B 0,C 180,E1 -20123.308,E2 -20123.308} C_VEL
LIN {X 0,Y 227.881,Z 89.1,A -85,B 0,C 180,E1 -20126.378,E2 -20126.378} C_VEL
LIN {X 0,Y 227.876,Z 89.1,A -85,B 0,C 180,E1 -20130.431,E2 -20130.431} C_VEL
LIN {X 0,Y 227.905,Z 89.095,A -85,B 0,C 180,E1 -20134.422,E2 -20134.422} C_VEL
LIN {X 0,Y 227.955,Z 89.08,A -85,B 0,C 180,E1 -20138.286,E2 -20138.286} C_VEL
LIN {X 0,Y 228.013,Z 89.068,A -85,B 0,C 180,E1 -20142.847,E2 -20142.847} C_VEL
LIN {X 0,Y 228.059,Z 89.06,A -85,B 0,C 180,E1 -20147.542,E2 -20147.542} C_VEL
LIN {X 0,Y 228.256,Z 89.052,A -85,B 0,C 180,E1 -20151.144,E2 -20151.144} C_VEL
LIN {X 0,Y 228.304,Z 89.031,A -85,B 0,C 180,E1 -20152.927,E2 -20152.927} C_VEL
LIN {X 0,Y 228.54,Z 89.009,A -85,B 0,C 180,E1 -20158.237,E2 -20158.237} C_VEL
LIN {X 0,Y 228.54,Z 89.011,A -85,B 0,C 180,E1 -20161.762,E2 -20161.762} C_VEL
LIN {X 0,Y 228.309,Z 89.032,A -85,B 0,C 180,E1 -20167.073,E2 -20167.073} C_VEL
LIN {X 0,Y 228.145,Z 89.053,A -85,B 0,C 180,E1 -20170.651,E2 -20170.651} C_VEL
LIN {X 0,Y 228.044,Z 89.078,A -85,B 0,C 180,E1 -20174.273,E2 -20174.273} C_VEL
LIN {X 0,Y 227.995,Z 89.07,A -85,B 0,C 180,E1 -20177.954,E2 -20177.954} C_VEL
LIN {X 0,Y 227.924,Z 89.082,A -85,B 0,C 180,E1 -20180.924,E2 -20180.924} C_VEL
LIN {X 0,Y 227.289,Z 89.16,A -85,B 0,C 180,E1 -20182.399,E2 -20182.399} C_VEL
LIN {X 0,Y 224.449,Z 89.528,A -85,B 0,C 180,E1 -20184.804,E2 -20184.804} C_VEL
LIN {X 0,Y 221.999,Z 89.838,A -85,B 0,C 180,E1 -20186.767,E2 -20186.767} C_VEL
LIN {X 0,Y 220.925,Z 89.966,A -85,B 0,C 180,E1 -20188.291,E2 -20188.291} C_VEL
LIN {X 0,Y 220.826,Z 89.974,A -85,B 0,C 180,E1 -20188.809,E2 -20188.809} C_VEL
LIN {X 0,Y 220.82,Z 89.979,A -85,B 0,C 180,E1 -20192.755,E2 -20192.755} C_VEL
LIN {X 0,Y 220.812,Z 89.946,A -85,B 0,C 180,E1 -20197.278,E2 -20197.278} C_VEL
LIN {X 0,Y 220.756,Z 90.009,A -85,B 0,C 180,E1 -20200.992,E2 -20200.992} C_VEL
LIN {X 0,Y 222.669,Z 96.435,A -85,B 0,C 180,E1 -20204.867,E2 -20204.867} C_VEL
LIN {X 0,Y 224.054,Z 101.187,A -85,B 0,C 180,E1 -20207.488,E2 -20207.488} C_VEL
LIN {X 0,Y 226.713,Z 105.854,A -85,B 0,C 180,E1 -20208.369,E2 -20208.369} C_VEL
LIN {X 0,Y 231.12,Z 113.512,A -85,B 0,C 180,E1 -20209.753,E2 -20209.753} C_VEL
LIN {X 0,Y 236.321,Z 123.312,A -85,B 0,C 180,E1 -20211.314,E2 -20211.314} C_VEL
LIN {X 0,Y 242.317,Z 135.953,A -85,B 0,C 180,E1 -20213.037,E2 -20213.037} C_VEL
LIN {X 0,Y 245.797,Z 144.405,A -85,B 0,C 180,E1 -20214.02,E2 -20214.02} C_VEL
LIN {X 0,Y 248.641,Z 164.05,A -85,B 0,C 180,E1 -20215.25,E2 -20215.25} C_VEL
LIN {X 0,Y 246.395,Z 211.287,A -85,B 0,C 180,E1 -20216.593,E2 -20216.593} C_VEL
LIN {X 0,Y 244.904,Z 224.941,A -85,B 0,C 180,E1 -20217.264,E2 -20217.264} C_VEL
LIN {X 0,Y 242.722,Z 237.997,A -85,B 0,C 180,E1 -20218.222,E2 -20218.222} C_VEL
LIN {X 0,Y 240.148,Z 249.81,A -85,B 0,C 180,E1 -20219.437,E2 -20219.437} C_VEL
LIN {X 0,Y 237.901,Z 258.604,A -85,B 0,C 180,E1 -20220.584,E2 -20220.584} C_VEL
LIN {X 0,Y 234.774,Z 269.321,A -85,B 0,C 180,E1 -20222.354,E2 -20222.354} C_VEL
LIN {X 0,Y 231.569,Z 278.984,A -85,B 0,C 180,E1 -20224.374,E2 -20224.374} C_VEL
LIN {X 0,Y 228.731,Z 286.922,A -85,B 0,C 180,E1 -20226.456,E2 -20226.456} C_VEL
LIN {X 0,Y 226.206,Z 293.965,A -85,B 0,C 180,E1 -20228.76,E2 -20228.76} C_VEL
LIN {X 0,Y 223.538,Z 300.983,A -85,B 0,C 180,E1 -20231.675,E2 -20231.675} C_VEL
LIN {X 0,Y 221.569,Z 305.988,A -85,B 0,C 180,E1 -20234.358,E2 -20234.358} C_VEL
LIN {X 0,Y 220.094,Z 309.879,A -85,B 0,C 180,E1 -20237.083,E2 -20237.083} C_VEL
LIN {X 0,Y 219.474,Z 311.899,A -85,B 0,C 180,E1 -20238.922,E2 -20238.922} C_VEL
LIN {X 0,Y 219.002,Z 313.511,A -85,B 0,C 180,E1 -20240.766,E2 -20240.766} C_VEL
LIN {X 0,Y 218.687,Z 314.712,A -85,B 0,C 180,E1 -20242.614,E2 -20242.614} C_VEL
LIN {X 0,Y 218.582,Z 315.865,A -85,B 0,C 180,E1 -20246.312,E2 -20246.312} C_VEL
LIN {X 0,Y 218.709,Z 315.865,A -85,B 0,C 180,E1 -20248.158,E2 -20248.158} C_VEL
LIN {X 0,Y 218.807,Z 315.47,A -85,B 0,C 180,E1 -20249.999,E2 -20249.999} C_VEL
LIN {X 0,Y 218.733,Z 314.622,A -85,B 0,C 180,E1 -20251.841,E2 -20251.841} C_VEL
LIN {X 0,Y 218.627,Z 312.428,A -85,B 0,C 180,E1 -20254.778,E2 -20254.778} C_VEL
LIN {X 0,Y 218.829,Z 308.313,A -85,B 0,C 180,E1 -20258.309,E2 -20258.309} C_VEL
LIN {X 0,Y 219.32,Z 303.842,A -85,B 0,C 180,E1 -20261.085,E2 -20261.085} C_VEL
LIN {X 0,Y 220.242,Z 298.158,A -85,B 0,C 180,E1 -20263.846,E2 -20263.846} C_VEL
LIN {X 0,Y 221.657,Z 291.039,A -85,B 0,C 180,E1 -20266.58,E2 -20266.58} C_VEL
LIN {X 0,Y 223.177,Z 284.105,A -85,B 0,C 180,E1 -20268.737,E2 -20268.737} C_VEL
LIN {X 0,Y 224.829,Z 274.953,A -85,B 0,C 180,E1 -20271.068,E2 -20271.068} C_VEL
LIN {X 0,Y 227.141,Z 264.125,A -85,B 0,C 180,E1 -20273.234,E2 -20273.234} C_VEL
LIN {X 0,Y 229.211,Z 253.304,A -85,B 0,C 180,E1 -20274.935,E2 -20274.935} C_VEL
LIN {X 0,Y 231.164,Z 241.13,A -85,B 0,C 180,E1 -20276.4,E2 -20276.4} C_VEL
LIN {X 0,Y 232.923,Z 228.43,A -85,B 0,C 180,E1 -20277.517,E2 -20277.517} C_VEL
LIN {X 0,Y 234,Z 215.893,A -85,B 0,C 180,E1 -20278.292,E2 -20278.292} C_VEL
LIN {X 0,Y 234.771,Z 199.557,A -85,B 0,C 180,E1 -20278.872,E2 -20278.872} C_VEL
LIN {X 0,Y 236.151,Z 158.158,A -85,B 0,C 180,E1 -20280.088,E2 -20280.088} C_VEL
LIN {X 0,Y 232.928,Z 130.027,A -85,B 0,C 180,E1 -20281.447,E2 -20281.447} C_VEL
LIN {X 0,Y 231.906,Z 122.747,A -85,B 0,C 180,E1 -20281.833,E2 -20281.833} C_VEL
LIN {X 0,Y 225.34,Z 106.343,A -85,B 0,C 180,E1 -20283.33,E2 -20283.33} C_VEL
LIN {X 0,Y 223.733,Z 102.414,A -85,B 0,C 180,E1 -20283.758,E2 -20283.758} C_VEL
LIN {X 0,Y 221.737,Z 93.622,A -85,B 0,C 180,E1 -20287.592,E2 -20287.592} C_VEL
LIN {X 0,Y 220.84,Z 89.98,A -85,B 0,C 180,E1 -20289.314,E2 -20289.314} C_VEL
LIN {X 0,Y 220.77,Z 89.985,A -85,B 0,C 180,E1 -20294.454,E2 -20294.454} C_VEL
LIN {X 0,Y 220.766,Z 89.985,A -85,B 0,C 180,E1 -20298.047,E2 -20298.047} C_VEL
LIN {X 0,Y 220.805,Z 89.961,A -85,B 0,C 180,E1 -20300.463,E2 -20300.463} C_VEL
LIN {X 0,Y 220.8,Z 89.98,A -85,B 0,C 180,E1 -20305.045,E2 -20305.045} C_VEL
LIN {X 0,Y 220.867,Z 89.973,A -85,B 0,C 180,E1 -20309.395,E2 -20309.395} C_VEL
LIN {X 0,Y 220.894,Z 89.961,A -85,B 0,C 180,E1 -20313.55,E2 -20313.55} C_VEL
LIN {X 0,Y 220.877,Z 89.968,A -85,B 0,C 180,E1 -20317.554,E2 -20317.554} C_VEL
LIN {X 0,Y 220.984,Z 89.957,A -85,B 0,C 180,E1 -20322.571,E2 -20322.571} C_VEL
LIN {X 0,Y 221.011,Z 89.939,A -85,B 0,C 180,E1 -20327.139,E2 -20327.139} C_VEL
LIN {X 0,Y 221.204,Z 89.93,A -85,B 0,C 180,E1 -20330.86,E2 -20330.86} C_VEL
LIN {X 0,Y 221.258,Z 89.923,A -85,B 0,C 180,E1 -20332.701,E2 -20332.701} C_VEL
LIN {X 0,Y 221.51,Z 89.886,A -85,B 0,C 180,E1 -20338.182,E2 -20338.182} C_VEL
LIN {X 0,Y 221.509,Z 89.891,A -85,B 0,C 180,E1 -20341.819,E2 -20341.819} C_VEL
LIN {X 0,Y 221.248,Z 89.919,A -85,B 0,C 180,E1 -20347.3,E2 -20347.3} C_VEL
LIN {X 0,Y 221.064,Z 89.942,A -85,B 0,C 180,E1 -20350.997,E2 -20350.997} C_VEL
LIN {X 0,Y 221.017,Z 89.95,A -85,B 0,C 180,E1 -20356.63,E2 -20356.63} C_VEL
LIN {X 0,Y 220.893,Z 89.958,A -85,B 0,C 180,E1 -20360.487,E2 -20360.487} C_VEL
LIN {X 0,Y 220.868,Z 89.969,A -85,B 0,C 180,E1 -20364.436,E2 -20364.436} C_VEL
LIN {X 0,Y 220.827,Z 89.975,A -85,B 0,C 180,E1 -20368.515,E2 -20368.515} C_VEL
LIN {X 0,Y 220.817,Z 89.979,A -85,B 0,C 180,E1 -20372.757,E2 -20372.757} C_VEL
LIN {X 0,Y 220.809,Z 89.979,A -85,B 0,C 180,E1 -20377.278,E2 -20377.278} C_VEL
LIN {X 0,Y 220.752,Z 89.985,A -85,B 0,C 180,E1 -20381.958,E2 -20381.958} C_VEL
LIN {X 0,Y 220.765,Z 89.985,A -85,B 0,C 180,E1 -20385.545,E2 -20385.545} C_VEL
LIN {X 0,Y 220.787,Z 89.982,A -85,B 0,C 180,E1 -20390.46,E2 -20390.46} C_VEL
LIN {X 0,Y 220.826,Z 89.978,A -85,B 0,C 180,E1 -20392.794,E2 -20392.794} C_VEL
LIN {X 0,Y 220.814,Z 89.974,A -85,B 0,C 180,E1 -20397.244,E2 -20397.244} C_VEL
LIN {X 0,Y 220.802,Z 89.965,A -85,B 0,C 180,E1 -20401.482,E2 -20401.482} C_VEL
LIN {X 0,Y 220.858,Z 89.972,A -85,B 0,C 180,E1 -20403.069,E2 -20403.069} C_VEL
LIN {X 0,Y 221.808,Z 92.701,A -85,B 0,C 180,E1 -20403.339,E2 -20403.339} C_VEL
LIN {X 0,Y 227.667,Z 103.59,A -85,B 0,C 180,E1 -20404.607,E2 -20404.607} C_VEL
LIN {X 0,Y 234.108,Z 117.108,A -85,B 0,C 180,E1 -20405.964,E2 -20405.964} C_VEL
LIN {X 0,Y 237.266,Z 125.971,A -85,B 0,C 180,E1 -20406.672,E2 -20406.672} C_VEL
LIN {X 0,Y 234.803,Z 192.739,A -85,B 0,C 180,E1 -20408.652,E2 -20408.652} C_VEL
LIN {X 0,Y 233.898,Z 205.971,A -85,B 0,C 180,E1 -20409.384,E2 -20409.384} C_VEL
LIN {X 0,Y 232.607,Z 219.069,A -85,B 0,C 180,E1 -20410.474,E2 -20410.474} C_VEL
LIN {X 0,Y 231.083,Z 230.883,A -85,B 0,C 180,E1 -20411.837,E2 -20411.837} C_VEL
LIN {X 0,Y 229.213,Z 242.23,A -85,B 0,C 180,E1 -20413.524,E2 -20413.524} C_VEL
LIN {X 0,Y 227.267,Z 252.47,A -85,B 0,C 180,E1 -20415.449,E2 -20415.449} C_VEL
LIN {X 0,Y 225.465,Z 260.853,A -85,B 0,C 180,E1 -20417.397,E2 -20417.397} C_VEL
LIN {X 0,Y 223.484,Z 269.93,A -85,B 0,C 180,E1 -20420.041,E2 -20420.041} C_VEL
LIN {X 0,Y 221.814,Z 277.247,A -85,B 0,C 180,E1 -20422.719,E2 -20422.719} C_VEL
LIN {X 0,Y 220.588,Z 283.114,A -85,B 0,C 180,E1 -20425.432,E2 -20425.432} C_VEL
LIN {X 0,Y 219.734,Z 287.748,A -85,B 0,C 180,E1 -20428.168,E2 -20428.168} C_VEL
LIN {X 0,Y 219.104,Z 291.296,A -85,B 0,C 180,E1 -20430.92,E2 -20430.92} C_VEL
LIN {X 0,Y 218.877,Z 293.841,A -85,B 0,C 180,E1 -20433.683,E2 -20433.683} C_VEL
LIN {X 0,Y 218.857,Z 295.042,A -85,B 0,C 180,E1 -20435.529,E2 -20435.529} C_VEL
LIN {X 0,Y 218.783,Z 295.814,A -85,B 0,C 180,E1 -20437.383,E2 -20437.383} C_VEL
LIN {X 0,Y 218.903,Z 296.196,A -85,B 0,C 180,E1 -20441.107,E2 -20441.107} C_VEL
LIN {X 0,Y 219.229,Z 295.806,A -85,B 0,C 180,E1 -20442.968,E2 -20442.968} C_VEL
LIN {X 0,Y 219.765,Z 294.974,A -85,B 0,C 180,E1 -20444.824,E2 -20444.824} C_VEL
LIN {X 0,Y 220.617,Z 293.394,A -85,B 0,C 180,E1 -20447.119,E2 -20447.119} C_VEL
LIN {X 0,Y 222.201,Z 290.01,A -85,B 0,C 180,E1 -20450.361,E2 -20450.361} C_VEL
LIN {X 0,Y 223.984,Z 285.963,A -85,B 0,C 180,E1 -20453.093,E2 -20453.093} C_VEL
LIN {X 0,Y 226.593,Z 279.706,A -85,B 0,C 180,E1 -20456.231,E2 -20456.231} C_VEL
LIN {X 0,Y 229.335,Z 272.859,A -85,B 0,C 180,E1 -20458.86,E2 -20458.86} C_VEL
LIN {X 0,Y 231.953,Z 265.838,A -85,B 0,C 180,E1 -20461.004,E2 -20461.004} C_VEL
LIN {X 0,Y 234.935,Z 256.704,A -85,B 0,C 180,E1 -20463.256,E2 -20463.256} C_VEL
LIN {X 0,Y 237.492,Z 247.953,A -85,B 0,C 180,E1 -20464.985,E2 -20464.985} C_VEL
LIN {X 0,Y 240.26,Z 237.705,A -85,B 0,C 180,E1 -20466.585,E2 -20466.585} C_VEL
LIN {X 0,Y 242.801,Z 226.581,A -85,B 0,C 180,E1 -20467.944,E2 -20467.944} C_VEL
LIN {X 0,Y 244.725,Z 214.982,A -85,B 0,C 180,E1 -20469.06,E2 -20469.06} C_VEL
LIN {X 0,Y 246.438,Z 202.045,A -85,B 0,C 180,E1 -20469.92,E2 -20469.92} C_VEL
LIN {X 0,Y 247.528,Z 188.781,A -85,B 0,C 180,E1 -20470.477,E2 -20470.477} C_VEL
LIN {X 0,Y 249.73,Z 140.29,A -85,B 0,C 180,E1 -20471.831,E2 -20471.831} C_VEL
LIN {X 0,Y 243.574,Z 126.766,A -85,B 0,C 180,E1 -20473.487,E2 -20473.487} C_VEL
LIN {X 0,Y 238.737,Z 117.829,A -85,B 0,C 180,E1 -20474.814,E2 -20474.814} C_VEL
LIN {X 0,Y 231.298,Z 106.21,A -85,B 0,C 180,E1 -20476.935,E2 -20476.935} C_VEL
LIN {X 0,Y 226.355,Z 98.941,A -85,B 0,C 180,E1 -20478.448,E2 -20478.448} C_VEL
LIN {X 0,Y 224.125,Z 95.594,A -85,B 0,C 180,E1 -20479.169,E2 -20479.169} C_VEL
LIN {X 0,Y 223.021,Z 94.326,A -85,B 0,C 180,E1 -20479.517,E2 -20479.517} C_VEL
LIN {X 0,Y 221.308,Z 91.936,A -85,B 0,C 180,E1 -20480.089,E2 -20480.089} C_VEL
LIN {X 0,Y 220.788,Z 89.982,A -85,B 0,C 180,E1 -20480.338,E2 -20480.338} C_VEL
LIN {X 0,Y 220.828,Z 89.978,A -85,B 0,C 180,E1 -20482.793,E2 -20482.793} C_VEL
LIN {X 0,Y 220.814,Z 89.975,A -85,B 0,C 180,E1 -20487.243,E2 -20487.243} C_VEL
LIN {X 0,Y 220.804,Z 89.974,A -85,B 0,C 180,E1 -20491.481,E2 -20491.481} C_VEL
LIN {X 0,Y 220.85,Z 89.973,A -85,B 0,C 180,E1 -20495.562,E2 -20495.562} C_VEL
LIN {X 0,Y 220.883,Z 89.972,A -85,B 0,C 180,E1 -20499.512,E2 -20499.512} C_VEL
LIN {X 0,Y 220.995,Z 89.944,A -85,B 0,C 180,E1 -20503.368,E2 -20503.368} C_VEL
LIN {X 0,Y 221.065,Z 89.934,A -85,B 0,C 180,E1 -20509.003,E2 -20509.003} C_VEL
LIN {X 0,Y 221.241,Z 89.912,A -85,B 0,C 180,E1 -20512.7,E2 -20512.7} C_VEL
LIN {X 0,Y 221.473,Z 89.889,A -85,B 0,C 180,E1 -20518.181,E2 -20518.181} C_VEL
LIN {X 0,Y 221.473,Z 89.892,A -85,B 0,C 180,E1 -20521.818,E2 -20521.818} C_VEL
LIN {X 0,Y 221.246,Z 89.913,A -85,B 0,C 180,E1 -20527.299,E2 -20527.299} C_VEL
LIN {X 0,Y 221.065,Z 89.931,A -85,B 0,C 180,E1 -20530.996,E2 -20530.996} C_VEL
LIN {X 0,Y 220.995,Z 89.941,A -85,B 0,C 180,E1 -20536.631,E2 -20536.631} C_VEL
LIN {X 0,Y 220.868,Z 89.965,A -85,B 0,C 180,E1 -20540.905,E2 -20540.905} C_VEL
LIN {X 0,Y 220.87,Z 89.973,A -85,B 0,C 180,E1 -20544.434,E2 -20544.434} C_VEL
LIN {X 0,Y 220.839,Z 89.975,A -85,B 0,C 180,E1 -20548.513,E2 -20548.513} C_VEL
LIN {X 0,Y 220.826,Z 89.974,A -85,B 0,C 180,E1 -20548.809,E2 -20548.809} C_VEL
LIN {X 0,Y 220.128,Z 90.06,A -85,B 0,C 180,E1 -20550.332,E2 -20550.332} C_VEL
LIN {X 0,Y 217.268,Z 90.421,A -85,B 0,C 180,E1 -20552.818,E2 -20552.818} C_VEL
LIN {X 0,Y 214.85,Z 90.7,A -85,B 0,C 180,E1 -20554.848,E2 -20554.848} C_VEL
LIN {X 0,Y 213.808,Z 90.816,A -85,B 0,C 180,E1 -20556.424,E2 -20556.424} C_VEL
LIN {X 0,Y 213.719,Z 90.827,A -85,B 0,C 180,E1 -20556.959,E2 -20556.959} C_VEL
LIN {X 0,Y 213.788,Z 91.041,A -85,B 0,C 180,E1 -20559.41,E2 -20559.41} C_VEL
LIN {X 0,Y 216.078,Z 98.731,A -85,B 0,C 180,E1 -20564.31,E2 -20564.31} C_VEL
LIN {X 0,Y 216.694,Z 100.792,A -85,B 0,C 180,E1 -20565.458,E2 -20565.458} C_VEL
LIN {X 0,Y 219.477,Z 105.457,A -85,B 0,C 180,E1 -20566.462,E2 -20566.462} C_VEL
LIN {X 0,Y 226.064,Z 116.59,A -85,B 0,C 180,E1 -20568.675,E2 -20568.675} C_VEL
LIN {X 0,Y 233.111,Z 130.249,A -85,B 0,C 180,E1 -20570.894,E2 -20570.894} C_VEL
LIN {X 0,Y 239.626,Z 144.803,A -85,B 0,C 180,E1 -20572.839,E2 -20572.839} C_VEL
LIN {X 0,Y 240.559,Z 147.585,A -85,B 0,C 180,E1 -20573.132,E2 -20573.132} C_VEL
LIN {X 0,Y 243.029,Z 165.022,A -85,B 0,C 180,E1 -20574.262,E2 -20574.262} C_VEL
LIN {X 0,Y 240.701,Z 211.2,A -85,B 0,C 180,E1 -20575.596,E2 -20575.596} C_VEL
LIN {X 0,Y 239.114,Z 225.188,A -85,B 0,C 180,E1 -20576.304,E2 -20576.304} C_VEL
LIN {X 0,Y 236.961,Z 237.546,A -85,B 0,C 180,E1 -20577.229,E2 -20577.229} C_VEL
LIN {X 0,Y 234.504,Z 248.6,A -85,B 0,C 180,E1 -20578.367,E2 -20578.367} C_VEL
LIN {X 0,Y 232.114,Z 257.542,A -85,B 0,C 180,E1 -20579.525,E2 -20579.525} C_VEL
LIN {X 0,Y 228.896,Z 268.398,A -85,B 0,C 180,E1 -20581.33,E2 -20581.33} C_VEL
LIN {X 0,Y 225.827,Z 277.27,A -85,B 0,C 180,E1 -20583.175,E2 -20583.175} C_VEL
LIN {X 0,Y 222.243,Z 286.925,A -85,B 0,C 180,E1 -20585.725,E2 -20585.725} C_VEL
LIN {X 0,Y 219.417,Z 294.357,A -85,B 0,C 180,E1 -20588.261,E2 -20588.261} C_VEL
LIN {X 0,Y 216.79,Z 300.857,A -85,B 0,C 180,E1 -20591.083,E2 -20591.083} C_VEL
LIN {X 0,Y 214.716,Z 305.819,A -85,B 0,C 180,E1 -20593.845,E2 -20593.845} C_VEL
LIN {X 0,Y 213.136,Z 309.67,A -85,B 0,C 180,E1 -20596.654,E2 -20596.654} C_VEL
LIN {X 0,Y 211.982,Z 313.267,A -85,B 0,C 180,E1 -20600.458,E2 -20600.458} C_VEL
LIN {X 0,Y 211.627,Z 314.435,A -85,B 0,C 180,E1 -20602.366,E2 -20602.366} C_VEL
LIN {X 0,Y 211.486,Z 315.552,A -85,B 0,C 180,E1 -20606.189,E2 -20606.189} C_VEL
LIN {X 0,Y 211.617,Z 315.536,A -85,B 0,C 180,E1 -20608.096,E2 -20608.096} C_VEL
LIN {X 0,Y 211.739,Z 315.115,A -85,B 0,C 180,E1 -20609.999,E2 -20609.999} C_VEL
LIN {X 0,Y 211.643,Z 314.241,A -85,B 0,C 180,E1 -20611.902,E2 -20611.902} C_VEL
LIN {X 0,Y 211.534,Z 312.288,A -85,B 0,C 180,E1 -20614.645,E2 -20614.645} C_VEL
LIN {X 0,Y 211.653,Z 309.117,A -85,B 0,C 180,E1 -20617.632,E2 -20617.632} C_VEL
LIN {X 0,Y 212.083,Z 304.983,A -85,B 0,C 180,E1 -20620.501,E2 -20620.501} C_VEL
LIN {X 0,Y 213.097,Z 298.639,A -85,B 0,C 180,E1 -20623.833,E2 -20623.833} C_VEL
LIN {X 0,Y 214.542,Z 291.735,A -85,B 0,C 180,E1 -20626.656,E2 -20626.656} C_VEL
LIN {X 0,Y 216.151,Z 284.688,A -85,B 0,C 180,E1 -20628.974,E2 -20628.974} C_VEL
LIN {X 0,Y 217.771,Z 276.164,A -85,B 0,C 180,E1 -20631.288,E2 -20631.288} C_VEL
LIN {X 0,Y 220.085,Z 265.663,A -85,B 0,C 180,E1 -20633.525,E2 -20633.525} C_VEL
LIN {X 0,Y 222.178,Z 255.264,A -85,B 0,C 180,E1 -20635.279,E2 -20635.279} C_VEL
LIN {X 0,Y 224.182,Z 243.862,A -85,B 0,C 180,E1 -20636.785,E2 -20636.785} C_VEL
LIN {X 0,Y 225.928,Z 232.201,A -85,B 0,C 180,E1 -20637.94,E2 -20637.94} C_VEL
LIN {X 0,Y 227.345,Z 218.723,A -85,B 0,C 180,E1 -20638.882,E2 -20638.882} C_VEL
LIN {X 0,Y 228.22,Z 205.428,A -85,B 0,C 180,E1 -20639.455,E2 -20639.455} C_VEL
LIN {X 0,Y 229.78,Z 158.618,A -85,B 0,C 180,E1 -20640.873,E2 -20640.873} C_VEL
LIN {X 0,Y 226.461,Z 128.986,A -85,B 0,C 180,E1 -20642.359,E2 -20642.359} C_VEL
LIN {X 0,Y 225.608,Z 124.429,A -85,B 0,C 180,E1 -20642.642,E2 -20642.642} C_VEL
LIN {X 0,Y 219.504,Z 109.289,A -85,B 0,C 180,E1 -20644.1,E2 -20644.1} C_VEL
LIN {X 0,Y 216.531,Z 102.11,A -85,B 0,C 180,E1 -20644.867,E2 -20644.867} C_VEL
LIN {X 0,Y 214.431,Z 93.37,A -85,B 0,C 180,E1 -20648.883,E2 -20648.883} C_VEL
LIN {X 0,Y 213.768,Z 90.858,A -85,B 0,C 180,E1 -20650.141,E2 -20650.141} C_VEL
LIN {X 0,Y 213.704,Z 90.867,A -85,B 0,C 180,E1 -20653.678,E2 -20653.678} C_VEL
LIN {X 0,Y 213.702,Z 90.866,A -85,B 0,C 180,E1 -20656.345,E2 -20656.345} C_VEL
LIN {X 0,Y 213.715,Z 90.855,A -85,B 0,C 180,E1 -20659.143,E2 -20659.143} C_VEL
LIN {X 0,Y 213.742,Z 90.852,A -85,B 0,C 180,E1 -20663.712,E2 -20663.712} C_VEL
LIN {X 0,Y 213.794,Z 90.854,A -85,B 0,C 180,E1 -20668.725,E2 -20668.725} C_VEL
LIN {X 0,Y 213.825,Z 90.843,A -85,B 0,C 180,E1 -20672.603,E2 -20672.603} C_VEL
LIN {X 0,Y 213.851,Z 90.846,A -85,B 0,C 180,E1 -20676.953,E2 -20676.953} C_VEL
LIN {X 0,Y 213.961,Z 90.833,A -85,B 0,C 180,E1 -20682.805,E2 -20682.805} C_VEL
LIN {X 0,Y 213.952,Z 90.819,A -85,B 0,C 180,E1 -20686.707,E2 -20686.707} C_VEL
LIN {X 0,Y 214.142,Z 90.809,A -85,B 0,C 180,E1 -20690.556,E2 -20690.556} C_VEL
LIN {X 0,Y 214.097,Z 90.808,A -85,B 0,C 180,E1 -20694.349,E2 -20694.349} C_VEL
LIN {X 0,Y 214.443,Z 90.766,A -85,B 0,C 180,E1 -20698.122,E2 -20698.122} C_VEL
LIN {X 0,Y 214.545,Z 90.76,A -85,B 0,C 180,E1 -20700,E2 -20700} C_VEL
LIN {X 0,Y 214.442,Z 90.77,A -85,B 0,C 180,E1 -20701.879,E2 -20701.879} C_VEL
LIN {X 0,Y 214.188,Z 90.8,A -85,B 0,C 180,E1 -20707.542,E2 -20707.542} C_VEL
LIN {X 0,Y 213.996,Z 90.82,A -85,B 0,C 180,E1 -20711.365,E2 -20711.365} C_VEL
LIN {X 0,Y 213.93,Z 90.828,A -85,B 0,C 180,E1 -20715.238,E2 -20715.238} C_VEL
LIN {X 0,Y 213.84,Z 90.842,A -85,B 0,C 180,E1 -20719.188,E2 -20719.188} C_VEL
LIN {X 0,Y 213.848,Z 90.839,A -85,B 0,C 180,E1 -20723.228,E2 -20723.228} C_VEL
LIN {X 0,Y 213.829,Z 90.847,A -85,B 0,C 180,E1 -20727.451,E2 -20727.451} C_VEL
LIN {X 0,Y 213.768,Z 90.856,A -85,B 0,C 180,E1 -20731.738,E2 -20731.738} C_VEL
LIN {X 0,Y 213.744,Z 90.86,A -85,B 0,C 180,E1 -20736.289,E2 -20736.289} C_VEL
LIN {X 0,Y 213.699,Z 90.865,A -85,B 0,C 180,E1 -20741.129,E2 -20741.129} C_VEL
LIN {X 0,Y 213.702,Z 90.865,A -85,B 0,C 180,E1 -20743.68,E2 -20743.68} C_VEL
LIN {X 0,Y 213.703,Z 90.867,A -85,B 0,C 180,E1 -20746.346,E2 -20746.346} C_VEL
LIN {X 0,Y 213.71,Z 90.864,A -85,B 0,C 180,E1 -20749.146,E2 -20749.146} C_VEL
LIN {X 0,Y 213.742,Z 90.86,A -85,B 0,C 180,E1 -20753.712,E2 -20753.712} C_VEL
LIN {X 0,Y 213.76,Z 90.857,A -85,B 0,C 180,E1 -20758.262,E2 -20758.262} C_VEL
LIN {X 0,Y 213.775,Z 90.921,A -85,B 0,C 180,E1 -20761.973,E2 -20761.973} C_VEL
LIN {X 0,Y 214.704,Z 93.576,A -85,B 0,C 180,E1 -20762.232,E2 -20762.232} C_VEL
LIN {X 0,Y 217.957,Z 99.178,A -85,B 0,C 180,E1 -20762.977,E2 -20762.977} C_VEL
LIN {X 0,Y 225.935,Z 114.934,A -85,B 0,C 180,E1 -20764.764,E2 -20764.764} C_VEL
LIN {X 0,Y 228.72,Z 121.209,A -85,B 0,C 180,E1 -20765.379,E2 -20765.379} C_VEL
LIN {X 0,Y 230.96,Z 127.654,A -85,B 0,C 180,E1 -20765.909,E2 -20765.909} C_VEL
LIN {X 0,Y 228.422,Z 193.143,A -85,B 0,C 180,E1 -20767.897,E2 -20767.897} C_VEL
LIN {X 0,Y 227.455,Z 206.464,A -85,B 0,C 180,E1 -20768.653,E2 -20768.653} C_VEL
LIN {X 0,Y 226.119,Z 219.509,A -85,B 0,C 180,E1 -20769.771,E2 -20769.771} C_VEL
LIN {X 0,Y 224.388,Z 232.08,A -85,B 0,C 180,E1 -20771.275,E2 -20771.275} C_VEL
LIN {X 0,Y 222.478,Z 243.264,A -85,B 0,C 180,E1 -20773.011,E2 -20773.011} C_VEL
LIN {X 0,Y 220.459,Z 253.356,A -85,B 0,C 180,E1 -20774.989,E2 -20774.989} C_VEL
LIN {X 0,Y 218.231,Z 263.256,A -85,B 0,C 180,E1 -20777.445,E2 -20777.445} C_VEL
LIN {X 0,Y 216.186,Z 271.976,A -85,B 0,C 180,E1 -20780.174,E2 -20780.174} C_VEL
LIN {X 0,Y 214.575,Z 278.945,A -85,B 0,C 180,E1 -20782.945,E2 -20782.945} C_VEL
LIN {X 0,Y 213.263,Z 285.314,A -85,B 0,C 180,E1 -20786.222,E2 -20786.222} C_VEL
LIN {X 0,Y 212.387,Z 289.528,A -85,B 0,C 180,E1 -20789.053,E2 -20789.053} C_VEL
LIN {X 0,Y 211.924,Z 292.687,A -85,B 0,C 180,E1 -20791.901,E2 -20791.901} C_VEL
LIN {X 0,Y 211.782,Z 295.257,A -85,B 0,C 180,E1 -20795.397,E2 -20795.397} C_VEL
LIN {X 0,Y 211.671,Z 296.172,A -85,B 0,C 180,E1 -20797.633,E2 -20797.633} C_VEL
LIN {X 0,Y 211.876,Z 296.508,A -85,B 0,C 180,E1 -20801.48,E2 -20801.48} C_VEL
LIN {X 0,Y 212.249,Z 296.082,A -85,B 0,C 180,E1 -20803.403,E2 -20803.403} C_VEL
LIN {X 0,Y 213.555,Z 293.96,A -85,B 0,C 180,E1 -20807.229,E2 -20807.229} C_VEL
LIN {X 0,Y 214.91,Z 291.27,A -85,B 0,C 180,E1 -20810.083,E2 -20810.083} C_VEL
LIN {X 0,Y 216.647,Z 287.542,A -85,B 0,C 180,E1 -20812.91,E2 -20812.91} C_VEL
LIN {X 0,Y 218.675,Z 283.063,A -85,B 0,C 180,E1 -20815.489,E2 -20815.489} C_VEL
LIN {X 0,Y 221.539,Z 276.482,A -85,B 0,C 180,E1 -20818.416,E2 -20818.416} C_VEL
LIN {X 0,Y 224.661,Z 268.734,A -85,B 0,C 180,E1 -20821.076,E2 -20821.076} C_VEL
LIN {X 0,Y 227.831,Z 259.915,A -85,B 0,C 180,E1 -20823.449,E2 -20823.449} C_VEL
LIN {X 0,Y 230.958,Z 249.911,A -85,B 0,C 180,E1 -20825.59,E2 -20825.59} C_VEL
LIN {X 0,Y 233.804,Z 240.088,A -85,B 0,C 180,E1 -20827.226,E2 -20827.226} C_VEL
LIN {X 0,Y 236.393,Z 229.375,A -85,B 0,C 180,E1 -20828.634,E2 -20828.634} C_VEL
LIN {X 0,Y 238.757,Z 216.801,A -85,B 0,C 180,E1 -20829.899,E2 -20829.899} C_VEL
LIN {X 0,Y 240.59,Z 204.037,A -85,B 0,C 180,E1 -20830.814,E2 -20830.814} C_VEL
LIN {X 0,Y 241.792,Z 191.282,A -85,B 0,C 180,E1 -20831.394,E2 -20831.394} C_VEL
LIN {X 0,Y 244.022,Z 142.361,A -85,B 0,C 180,E1 -20832.816,E2 -20832.816} C_VEL
LIN {X 0,Y 237.911,Z 129.043,A -85,B 0,C 180,E1 -20834.547,E2 -20834.547} C_VEL
LIN {X 0,Y 233.179,Z 120.543,A -85,B 0,C 180,E1 -20835.911,E2 -20835.911} C_VEL
LIN {X 0,Y 225.373,Z 108.299,A -85,B 0,C 180,E1 -20838.283,E2 -20838.283} C_VEL
LIN {X 0,Y 219.565,Z 99.976,A -85,B 0,C 180,E1 -20840.194,E2 -20840.194} C_VEL
LIN {X 0,Y 217.324,Z 96.763,A -85,B 0,C 180,E1 -20840.979,E2 -20840.979} C_VEL
LIN {X 0,Y 216.679,Z 95.76,A -85,B 0,C 180,E1 -20841.214,E2 -20841.214} C_VEL
LIN {X 0,Y 214.621,Z 93.544,A -85,B 0,C 180,E1 -20841.931,E2 -20841.931} C_VEL
LIN {X 0,Y 213.747,Z 90.856,A -85,B 0,C 180,E1 -20842.362,E2 -20842.362} C_VEL
LIN {X 0,Y 213.757,Z 90.856,A -85,B 0,C 180,E1 -20846.017,E2 -20846.017} C_VEL
LIN {X 0,Y 213.752,Z 90.86,A -85,B 0,C 180,E1 -20850.449,E2 -20850.449} C_VEL
LIN {X 0,Y 213.785,Z 90.855,A -85,B 0,C 180,E1 -20854.699,E2 -20854.699} C_VEL
LIN {X 0,Y 213.804,Z 90.847,A -85,B 0,C 180,E1 -20858.802,E2 -20858.802} C_VEL
LIN {X 0,Y 213.925,Z 90.821,A -85,B 0,C 180,E1 -20862.802,E2 -20862.802} C_VEL
LIN {X 0,Y 213.94,Z 90.824,A -85,B 0,C 180,E1 -20866.705,E2 -20866.705} C_VEL
LIN {X 0,Y 214.137,Z 90.811,A -85,B 0,C 180,E1 -20870.555,E2 -20870.555} C_VEL
LIN {X 0,Y 214.08,Z 90.799,A -85,B 0,C 180,E1 -20874.348,E2 -20874.348} C_VEL
LIN {X 0,Y 214.41,Z 90.769,A -85,B 0,C 180,E1 -20878.121,E2 -20878.121} C_VEL
LIN {X 0,Y 214.515,Z 90.744,A -85,B 0,C 180,E1 -20880,E2 -20880} C_VEL
LIN {X 0,Y 214.41,Z 90.772,A -85,B 0,C 180,E1 -20881.878,E2 -20881.878} C_VEL
LIN {X 0,Y 214.188,Z 90.795,A -85,B 0,C 180,E1 -20887.541,E2 -20887.541} C_VEL
LIN {X 0,Y 213.997,Z 90.809,A -85,B 0,C 180,E1 -20891.364,E2 -20891.364} C_VEL
LIN {X 0,Y 213.912,Z 90.834,A -85,B 0,C 180,E1 -20895.238,E2 -20895.238} C_VEL
LIN {X 0,Y 213.837,Z 90.845,A -85,B 0,C 180,E1 -20899.187,E2 -20899.187} C_VEL
LIN {X 0,Y 213.85,Z 90.835,A -85,B 0,C 180,E1 -20903.226,E2 -20903.226} C_VEL
LIN {X 0,Y 213.832,Z 90.838,A -85,B 0,C 180,E1 -20907.449,E2 -20907.449} C_VEL
LIN {X 0,Y 213.779,Z 90.847,A -85,B 0,C 180,E1 -20911.735,E2 -20911.735} C_VEL
LIN {X 0,Y 213.746,Z 90.823,A -85,B 0,C 180,E1 -20916.288,E2 -20916.288} C_VEL
LIN {X 0,Y 213.719,Z 90.827,A -85,B 0,C 180,E1 -20916.959,E2 -20916.959} C_VEL
LIN {X 0,Y 213.156,Z 91.345,A -85,B 0,C 180,E1 -20917.999,E2 -20917.999} C_VEL
LIN {X 0,Y 210.93,Z 93.695,A -85,B 0,C 180,E1 -20919.589,E2 -20919.589} C_VEL
LIN {X 0,Y 208.91,Z 96.848,A -85,B 0,C 180,E1 -20921.161,E2 -20921.161} C_VEL
LIN {X 0,Y 208.734,Z 98.618,A -85,B 0,C 180,E1 -20922.165,E2 -20922.165} C_VEL
LIN {X 0,Y 209.292,Z 100.261,A -85,B 0,C 180,E1 -20923.172,E2 -20923.172} C_VEL
LIN {X 0,Y 211.921,Z 104.715,A -85,B 0,C 180,E1 -20924.229,E2 -20924.229} C_VEL
LIN {X 0,Y 213.384,Z 106.89,A -85,B 0,C 180,E1 -20924.782,E2 -20924.782} C_VEL
LIN {X 0,Y 216.926,Z 112.776,A -85,B 0,C 180,E1 -20926.097,E2 -20926.097} C_VEL
LIN {X 0,Y 222.02,Z 121.615,A -85,B 0,C 180,E1 -20927.878,E2 -20927.878} C_VEL
LIN {X 0,Y 228.548,Z 134.47,A -85,B 0,C 180,E1 -20930.034,E2 -20930.034} C_VEL
LIN {X 0,Y 234.839,Z 148.821,A -85,B 0,C 180,E1 -20932.013,E2 -20932.013} C_VEL
LIN {X 0,Y 235.489,Z 151.381,A -85,B 0,C 180,E1 -20932.25,E2 -20932.25} C_VEL
LIN {X 0,Y 237.441,Z 166.43,A -85,B 0,C 180,E1 -20933.234,E2 -20933.234} C_VEL
LIN {X 0,Y 235.111,Z 210.963,A -85,B 0,C 180,E1 -20934.548,E2 -20934.548} C_VEL
LIN {X 0,Y 233.49,Z 224.679,A -85,B 0,C 180,E1 -20935.248,E2 -20935.248} C_VEL
LIN {X 0,Y 231.287,Z 237.091,A -85,B 0,C 180,E1 -20936.188,E2 -20936.188} C_VEL
LIN {X 0,Y 228.519,Z 248.968,A -85,B 0,C 180,E1 -20937.438,E2 -20937.438} C_VEL
LIN {X 0,Y 226.018,Z 257.801,A -85,B 0,C 180,E1 -20938.611,E2 -20938.611} C_VEL
LIN {X 0,Y 222.705,Z 268.544,A -85,B 0,C 180,E1 -20940.456,E2 -20940.456} C_VEL
LIN {X 0,Y 218.868,Z 279.118,A -85,B 0,C 180,E1 -20942.768,E2 -20942.768} C_VEL
LIN {X 0,Y 215.203,Z 288.283,A -85,B 0,C 180,E1 -20945.393,E2 -20945.393} C_VEL
LIN {X 0,Y 212.118,Z 295.992,A -85,B 0,C 180,E1 -20948.255,E2 -20948.255} C_VEL
LIN {X 0,Y 209.286,Z 302.526,A -85,B 0,C 180,E1 -20951.396,E2 -20951.396} C_VEL
LIN {X 0,Y 207.275,Z 307.062,A -85,B 0,C 180,E1 -20954.261,E2 -20954.261} C_VEL
LIN {X 0,Y 206.197,Z 309.464,A -85,B 0,C 180,E1 -20956.196,E2 -20956.196} C_VEL
LIN {X 0,Y 204.944,Z 313.022,A -85,B 0,C 180,E1 -20960.127,E2 -20960.127} C_VEL
LIN {X 0,Y 204.394,Z 314.889,A -85,B 0,C 180,E1 -20964.079,E2 -20964.079} C_VEL
LIN {X 0,Y 204.404,Z 315.24,A -85,B 0,C 180,E1 -20966.056,E2 -20966.056} C_VEL
LIN {X 0,Y 204.528,Z 315.207,A -85,B 0,C 180,E1 -20968.03,E2 -20968.03} C_VEL
LIN {X 0,Y 204.671,Z 314.754,A -85,B 0,C 180,E1 -20969.999,E2 -20969.999} C_VEL
LIN {X 0,Y 204.556,Z 313.861,A -85,B 0,C 180,E1 -20971.968,E2 -20971.968} C_VEL
LIN {X 0,Y 204.466,Z 312.073,A -85,B 0,C 180,E1 -20974.584,E2 -20974.584} C_VEL
LIN {X 0,Y 204.607,Z 308.662,A -85,B 0,C 180,E1 -20977.897,E2 -20977.897} C_VEL
LIN {X 0,Y 205.064,Z 304.485,A -85,B 0,C 180,E1 -20980.865,E2 -20980.865} C_VEL
LIN {X 0,Y 206.172,Z 298.097,A -85,B 0,C 180,E1 -20984.308,E2 -20984.308} C_VEL
LIN {X 0,Y 207.688,Z 291.141,A -85,B 0,C 180,E1 -20987.222,E2 -20987.222} C_VEL
LIN {X 0,Y 209.349,Z 284.035,A -85,B 0,C 180,E1 -20989.615,E2 -20989.615} C_VEL
LIN {X 0,Y 211.094,Z 275.425,A -85,B 0,C 180,E1 -20991.996,E2 -20991.996} C_VEL
LIN {X 0,Y 213.553,Z 264.823,A -85,B 0,C 180,E1 -20994.291,E2 -20994.291} C_VEL
LIN {X 0,Y 215.77,Z 254.318,A -85,B 0,C 180,E1 -20996.085,E2 -20996.085} C_VEL
LIN {X 0,Y 217.853,Z 242.745,A -85,B 0,C 180,E1 -20997.628,E2 -20997.628} C_VEL
LIN {X 0,Y 219.72,Z 230.75,A -85,B 0,C 180,E1 -20998.802,E2 -20998.802} C_VEL
LIN {X 0,Y 221.057,Z 217.715,A -85,B 0,C 180,E1 -20999.72,E2 -20999.72} C_VEL
LIN {X 0,Y 221.861,Z 205.484,A -85,B 0,C 180,E1 -21000.256,E2 -21000.256} C_VEL
LIN {X 0,Y 223.504,Z 159.415,A -85,B 0,C 180,E1 -21001.683,E2 -21001.683} C_VEL
LIN {X 0,Y 220.283,Z 130.179,A -85,B 0,C 180,E1 -21003.207,E2 -21003.207} C_VEL
LIN {X 0,Y 219.568,Z 126.681,A -85,B 0,C 180,E1 -21003.443,E2 -21003.443} C_VEL
LIN {X 0,Y 213.816,Z 112.434,A -85,B 0,C 180,E1 -21004.885,E2 -21004.885} C_VEL
LIN {X 0,Y 210.533,Z 104.965,A -85,B 0,C 180,E1 -21005.728,E2 -21005.728} C_VEL
LIN {X 0,Y 209.186,Z 101.797,A -85,B 0,C 180,E1 -21006.089,E2 -21006.089} C_VEL
LIN {X 0,Y 207.142,Z 93.441,A -85,B 0,C 180,E1 -21010.138,E2 -21010.138} C_VEL
LIN {X 0,Y 206.689,Z 91.741,A -85,B 0,C 180,E1 -21011.038,E2 -21011.038} C_VEL
LIN {X 0,Y 206.63,Z 91.747,A -85,B 0,C 180,E1 -21015.582,E2 -21015.582} C_VEL
LIN {X 0,Y 206.659,Z 91.727,A -85,B 0,C 180,E1 -21019.748,E2 -21019.748} C_VEL
LIN {X 0,Y 206.698,Z 91.735,A -85,B 0,C 180,E1 -21024.689,E2 -21024.689} C_VEL
LIN {X 0,Y 206.722,Z 91.734,A -85,B 0,C 180,E1 -21029.339,E2 -21029.339} C_VEL
LIN {X 0,Y 206.732,Z 91.725,A -85,B 0,C 180,E1 -21033.772,E2 -21033.772} C_VEL
LIN {X 0,Y 206.757,Z 91.727,A -85,B 0,C 180,E1 -21038.044,E2 -21038.044} C_VEL
LIN {X 0,Y 206.873,Z 91.712,A -85,B 0,C 180,E1 -21042.197,E2 -21042.197} C_VEL
LIN {X 0,Y 206.895,Z 91.701,A -85,B 0,C 180,E1 -21046.245,E2 -21046.245} C_VEL
LIN {X 0,Y 207.098,Z 91.683,A -85,B 0,C 180,E1 -21050.231,E2 -21050.231} C_VEL
LIN {X 0,Y 207.059,Z 91.686,A -85,B 0,C 180,E1 -21054.156,E2 -21054.156} C_VEL
LIN {X 0,Y 207.379,Z 91.644,A -85,B 0,C 180,E1 -21058.058,E2 -21058.058} C_VEL
LIN {X 0,Y 207.511,Z 91.636,A -85,B 0,C 180,E1 -21060,E2 -21060} C_VEL
LIN {X 0,Y 207.378,Z 91.649,A -85,B 0,C 180,E1 -21061.943,E2 -21061.943} C_VEL
LIN {X 0,Y 207.132,Z 91.68,A -85,B 0,C 180,E1 -21067.801,E2 -21067.801} C_VEL
LIN {X 0,Y 206.92,Z 91.697,A -85,B 0,C 180,E1 -21071.759,E2 -21071.759} C_VEL
LIN {X 0,Y 206.864,Z 91.711,A -85,B 0,C 180,E1 -21075.771,E2 -21075.771} C_VEL
LIN {X 0,Y 206.784,Z 91.715,A -85,B 0,C 180,E1 -21079.87,E2 -21079.87} C_VEL
LIN {X 0,Y 206.764,Z 91.726,A -85,B 0,C 180,E1 -21084.073,E2 -21084.073} C_VEL
LIN {X 0,Y 206.737,Z 91.73,A -85,B 0,C 180,E1 -21088.42,E2 -21088.42} C_VEL
LIN {X 0,Y 206.699,Z 91.739,A -85,B 0,C 180,E1 -21092.958,E2 -21092.958} C_VEL
LIN {X 0,Y 206.673,Z 91.739,A -85,B 0,C 180,E1 -21097.742,E2 -21097.742} C_VEL
LIN {X 0,Y 206.632,Z 91.744,A -85,B 0,C 180,E1 -21101.56,E2 -21101.56} C_VEL
LIN {X 0,Y 206.631,Z 91.746,A -85,B 0,C 180,E1 -21105.583,E2 -21105.583} C_VEL
LIN {X 0,Y 206.653,Z 91.743,A -85,B 0,C 180,E1 -21109.748,E2 -21109.748} C_VEL
LIN {X 0,Y 206.701,Z 91.737,A -85,B 0,C 180,E1 -21114.69,E2 -21114.69} C_VEL
LIN {X 0,Y 206.697,Z 91.734,A -85,B 0,C 180,E1 -21119.335,E2 -21119.335} C_VEL
LIN {X 0,Y 206.717,Z 91.718,A -85,B 0,C 180,E1 -21120.754,E2 -21120.754} C_VEL
LIN {X 0,Y 207.661,Z 94.484,A -85,B 0,C 180,E1 -21121.046,E2 -21121.046} C_VEL
LIN {X 0,Y 209.41,Z 97.425,A -85,B 0,C 180,E1 -21121.476,E2 -21121.476} C_VEL
LIN {X 0,Y 215.186,Z 107.748,A -85,B 0,C 180,E1 -21122.857,E2 -21122.857} C_VEL
LIN {X 0,Y 222.632,Z 123.375,A -85,B 0,C 180,E1 -21124.59,E2 -21124.59} C_VEL
LIN {X 0,Y 224.692,Z 129.402,A -85,B 0,C 180,E1 -21125.105,E2 -21125.105} C_VEL
LIN {X 0,Y 222.066,Z 193.941,A -85,B 0,C 180,E1 -21127.119,E2 -21127.119} C_VEL
LIN {X 0,Y 220.984,Z 207.707,A -85,B 0,C 180,E1 -21127.934,E2 -21127.934} C_VEL
LIN {X 0,Y 219.674,Z 219.94,A -85,B 0,C 180,E1 -21129.028,E2 -21129.028} C_VEL
LIN {X 0,Y 217.997,Z 231.699,A -85,B 0,C 180,E1 -21130.46,E2 -21130.46} C_VEL
LIN {X 0,Y 215.988,Z 243.012,A -85,B 0,C 180,E1 -21132.239,E2 -21132.239} C_VEL
LIN {X 0,Y 213.878,Z 253.226,A -85,B 0,C 180,E1 -21134.271,E2 -21134.271} C_VEL
LIN {X 0,Y 211.707,Z 262.41,A -85,B 0,C 180,E1 -21136.563,E2 -21136.563} C_VEL
LIN {X 0,Y 209.553,Z 271.322,A -85,B 0,C 180,E1 -21139.371,E2 -21139.371} C_VEL
LIN {X 0,Y 207.802,Z 278.506,A -85,B 0,C 180,E1 -21142.226,E2 -21142.226} C_VEL
LIN {X 0,Y 206.499,Z 284.249,A -85,B 0,C 180,E1 -21145.12,E2 -21145.12} C_VEL
LIN {X 0,Y 205.547,Z 288.777,A -85,B 0,C 180,E1 -21148.041,E2 -21148.041} C_VEL
LIN {X 0,Y 205.074,Z 291.171,A -85,B 0,C 180,E1 -21150.001,E2 -21150.001} C_VEL
LIN {X 0,Y 204.844,Z 293.13,A -85,B 0,C 180,E1 -21151.967,E2 -21151.967} C_VEL
LIN {X 0,Y 204.705,Z 295.519,A -85,B 0,C 180,E1 -21155.346,E2 -21155.346} C_VEL
LIN {X 0,Y 204.589,Z 296.528,A -85,B 0,C 180,E1 -21157.898,E2 -21157.898} C_VEL
LIN {X 0,Y 204.839,Z 296.821,A -85,B 0,C 180,E1 -21161.88,E2 -21161.88} C_VEL
LIN {X 0,Y 205.285,Z 296.35,A -85,B 0,C 180,E1 -21163.866,E2 -21163.866} C_VEL
LIN {X 0,Y 206.669,Z 294.183,A -85,B 0,C 180,E1 -21167.822,E2 -21167.822} C_VEL
LIN {X 0,Y 208.149,Z 291.445,A -85,B 0,C 180,E1 -21170.765,E2 -21170.765} C_VEL
LIN {X 0,Y 210.016,Z 287.666,A -85,B 0,C 180,E1 -21173.677,E2 -21173.677} C_VEL
LIN {X 0,Y 212.628,Z 282.192,A -85,B 0,C 180,E1 -21176.818,E2 -21176.818} C_VEL
LIN {X 0,Y 215.758,Z 275.289,A -85,B 0,C 180,E1 -21179.786,E2 -21179.786} C_VEL
LIN {X 0,Y 219.126,Z 267.145,A -85,B 0,C 180,E1 -21182.495,E2 -21182.495} C_VEL
LIN {X 0,Y 222.15,Z 258.787,A -85,B 0,C 180,E1 -21184.713,E2 -21184.713} C_VEL
LIN {X 0,Y 225.126,Z 249.628,A -85,B 0,C 180,E1 -21186.659,E2 -21186.659} C_VEL
LIN {X 0,Y 228.11,Z 239.628,A -85,B 0,C 180,E1 -21188.32,E2 -21188.32} C_VEL
LIN {X 0,Y 230.828,Z 228.705,A -85,B 0,C 180,E1 -21189.747,E2 -21189.747} C_VEL
LIN {X 0,Y 233.013,Z 217.424,A -85,B 0,C 180,E1 -21190.894,E2 -21190.894} C_VEL
LIN {X 0,Y 234.959,Z 204.314,A -85,B 0,C 180,E1 -21191.854,E2 -21191.854} C_VEL
LIN {X 0,Y 236.217,Z 191.172,A -85,B 0,C 180,E1 -21192.457,E2 -21192.457} C_VEL
LIN {X 0,Y 238.43,Z 144.429,A -85,B 0,C 180,E1 -21193.841,E2 -21193.841} C_VEL
LIN {X 0,Y 231.996,Z 130.605,A -85,B 0,C 180,E1 -21195.764,E2 -21195.764} C_VEL
LIN {X 0,Y 223.955,Z 117.163,A -85,B 0,C 180,E1 -21198.25,E2 -21198.25} C_VEL
LIN {X 0,Y 218.009,Z 108.432,A -85,B 0,C 180,E1 -21200.229,E2 -21200.229} C_VEL
LIN {X 0,Y 215.242,Z 104.539,A -85,B 0,C 180,E1 -21201.207,E2 -21201.207} C_VEL
LIN {X 0,Y 213.043,Z 101.325,A -85,B 0,C 180,E1 -21202.021,E2 -21202.021} C_VEL
LIN {X 0,Y 210.682,Z 98.188,A -85,B 0,C 180,E1 -21202.914,E2 -21202.914} C_VEL
LIN {X 0,Y 209.898,Z 96.81,A -85,B 0,C 180,E1 -21203.236,E2 -21203.236} C_VEL
LIN {X 0,Y 207.72,Z 94.61,A -85,B 0,C 180,E1 -21204.068,E2 -21204.068} C_VEL
LIN {X 0,Y 206.822,Z 92.458,A -85,B 0,C 180,E1 -21204.488,E2 -21204.488} C_VEL
LIN {X 0,Y 206.7,Z 91.729,A -85,B 0,C 180,E1 -21204.613,E2 -21204.613} C_VEL
LIN {X 0,Y 206.698,Z 91.73,A -85,B 0,C 180,E1 -21209.334,E2 -21209.334} C_VEL
LIN {X 0,Y 206.707,Z 91.729,A -85,B 0,C 180,E1 -21213.768,E2 -21213.768} C_VEL
LIN {X 0,Y 206.737,Z 91.72,A -85,B 0,C 180,E1 -21218.04,E2 -21218.04} C_VEL
LIN {X 0,Y 206.871,Z 91.7,A -85,B 0,C 180,E1 -21222.196,E2 -21222.196} C_VEL
LIN {X 0,Y 206.882,Z 91.707,A -85,B 0,C 180,E1 -21226.243,E2 -21226.243} C_VEL
LIN {X 0,Y 207.082,Z 91.688,A -85,B 0,C 180,E1 -21230.23,E2 -21230.23} C_VEL
LIN {X 0,Y 207.043,Z 91.675,A -85,B 0,C 180,E1 -21234.155,E2 -21234.155} C_VEL
LIN {X 0,Y 207.35,Z 91.649,A -85,B 0,C 180,E1 -21238.057,E2 -21238.057} C_VEL
LIN {X 0,Y 207.483,Z 91.619,A -85,B 0,C 180,E1 -21240,E2 -21240} C_VEL
LIN {X 0,Y 207.349,Z 91.652,A -85,B 0,C 180,E1 -21241.942,E2 -21241.942} C_VEL
LIN {X 0,Y 207.132,Z 91.676,A -85,B 0,C 180,E1 -21247.8,E2 -21247.8} C_VEL
LIN {X 0,Y 206.92,Z 91.69,A -85,B 0,C 180,E1 -21251.758,E2 -21251.758} C_VEL
LIN {X 0,Y 206.847,Z 91.709,A -85,B 0,C 180,E1 -21255.772,E2 -21255.772} C_VEL
LIN {X 0,Y 206.783,Z 91.727,A -85,B 0,C 180,E1 -21259.869,E2 -21259.869} C_VEL
LIN {X 0,Y 206.767,Z 91.726,A -85,B 0,C 180,E1 -21264.071,E2 -21264.071} C_VEL
LIN {X 0,Y 206.747,Z 91.729,A -85,B 0,C 180,E1 -21268.418,E2 -21268.418} C_VEL
LIN {X 0,Y 206.704,Z 91.738,A -85,B 0,C 180,E1 -21272.956,E2 -21272.956} C_VEL
LIN {X 0,Y 206.692,Z 91.768,A -85,B 0,C 180,E1 -21277.43,E2 -21277.43} C_VEL
LIN {X 0,Y 208.478,Z 97.697,A -85,B 0,C 180,E1 -21281.567,E2 -21281.567} C_VEL
LIN {X 0,Y 208.734,Z 98.618,A -85,B 0,C 180,E1 -21282.165,E2 -21282.165} C_VEL
LIN {X 0,Y 209.429,Z 100.658,A -85,B 0,C 180,E1 -21283.027,E2 -21283.027} C_VEL
LIN {X 0,Y 210.73,Z 104.249,A -85,B 0,C 180,E1 -21283.836,E2 -21283.836} C_VEL
LIN {X 0,Y 212.484,Z 110.226,A -85,B 0,C 180,E1 -21284.677,E2 -21284.677} C_VEL
LIN {X 0,Y 214.286,Z 117.685,A -85,B 0,C 180,E1 -21285.555,E2 -21285.555} C_VEL
LIN {X 0,Y 216.046,Z 122.861,A -85,B 0,C 180,E1 -21286.326,E2 -21286.326} C_VEL
LIN {X 0,Y 216.842,Z 124.396,A -85,B 0,C 180,E1 -21286.623,E2 -21286.623} C_VEL
LIN {X 0,Y 222.439,Z 135.357,A -85,B 0,C 180,E1 -21288.597,E2 -21288.597} C_VEL
LIN {X 0,Y 227.282,Z 146.037,A -85,B 0,C 180,E1 -21290.228,E2 -21290.228} C_VEL
LIN {X 0,Y 230.196,Z 153.273,A -85,B 0,C 180,E1 -21291.189,E2 -21291.189} C_VEL
LIN {X 0,Y 231.996,Z 167.114,A -85,B 0,C 180,E1 -21292.14,E2 -21292.14} C_VEL
LIN {X 0,Y 229.608,Z 210.658,A -85,B 0,C 180,E1 -21293.445,E2 -21293.445} C_VEL
LIN {X 0,Y 227.965,Z 224.178,A -85,B 0,C 180,E1 -21294.143,E2 -21294.143} C_VEL
LIN {X 0,Y 225.672,Z 236.643,A -85,B 0,C 180,E1 -21295.092,E2 -21295.092} C_VEL
LIN {X 0,Y 223.001,Z 247.764,A -85,B 0,C 180,E1 -21296.257,E2 -21296.257} C_VEL
LIN {X 0,Y 220.007,Z 258.045,A -85,B 0,C 180,E1 -21297.651,E2 -21297.651} C_VEL
LIN {X 0,Y 216.555,Z 268.69,A -85,B 0,C 180,E1 -21299.529,E2 -21299.529} C_VEL
LIN {X 0,Y 212.588,Z 279.169,A -85,B 0,C 180,E1 -21301.894,E2 -21301.894} C_VEL
LIN {X 0,Y 208.76,Z 288.258,A -85,B 0,C 180,E1 -21304.58,E2 -21304.58} C_VEL
LIN {X 0,Y 205.8,Z 295.224,A -85,B 0,C 180,E1 -21307.226,E2 -21307.226} C_VEL
LIN {X 0,Y 203.39,Z 300.61,A -85,B 0,C 180,E1 -21309.784,E2 -21309.784} C_VEL
LIN {X 0,Y 201.082,Z 305.487,A -85,B 0,C 180,E1 -21312.717,E2 -21312.717} C_VEL
LIN {X 0,Y 199.271,Z 309.258,A -85,B 0,C 180,E1 -21315.706,E2 -21315.706} C_VEL
LIN {X 0,Y 198.503,Z 311.223,A -85,B 0,C 180,E1 -21317.735,E2 -21317.735} C_VEL
LIN {X 0,Y 197.926,Z 312.773,A -85,B 0,C 180,E1 -21319.773,E2 -21319.773} C_VEL
LIN {X 0,Y 197.331,Z 314.594,A -85,B 0,C 180,E1 -21323.866,E2 -21323.866} C_VEL
LIN {X 0,Y 197.325,Z 314.928,A -85,B 0,C 180,E1 -21325.915,E2 -21325.915} C_VEL
LIN {X 0,Y 197.44,Z 314.876,A -85,B 0,C 180,E1 -21327.959,E2 -21327.959} C_VEL
LIN {X 0,Y 197.582,Z 314.39,A -85,B 0,C 180,E1 -21329.999,E2 -21329.999} C_VEL
LIN {X 0,Y 197.47,Z 313.479,A -85,B 0,C 180,E1 -21332.039,E2 -21332.039} C_VEL
LIN {X 0,Y 197.371,Z 311.92,A -85,B 0,C 180,E1 -21334.422,E2 -21334.422} C_VEL
LIN {X 0,Y 197.554,Z 308.204,A -85,B 0,C 180,E1 -21338.18,E2 -21338.18} C_VEL
LIN {X 0,Y 198.065,Z 303.986,A -85,B 0,C 180,E1 -21341.253,E2 -21341.253} C_VEL
LIN {X 0,Y 199.273,Z 297.554,A -85,B 0,C 180,E1 -21344.814,E2 -21344.814} C_VEL
LIN {X 0,Y 200.879,Z 290.543,A -85,B 0,C 180,E1 -21347.826,E2 -21347.826} C_VEL
LIN {X 0,Y 202.574,Z 283.374,A -85,B 0,C 180,E1 -21350.299,E2 -21350.299} C_VEL
LIN {X 0,Y 204.48,Z 274.674,A -85,B 0,C 180,E1 -21352.746,E2 -21352.746} C_VEL
LIN {X 0,Y 206.797,Z 265.168,A -85,B 0,C 180,E1 -21354.87,E2 -21354.87} C_VEL
LIN {X 0,Y 209.086,Z 254.805,A -85,B 0,C 180,E1 -21356.716,E2 -21356.716} C_VEL
LIN {X 0,Y 211.237,Z 243.446,A -85,B 0,C 180,E1 -21358.301,E2 -21358.301} C_VEL
LIN {X 0,Y 213.119,Z 231.88,A -85,B 0,C 180,E1 -21359.511,E2 -21359.511} C_VEL
LIN {X 0,Y 214.621,Z 218.539,A -85,B 0,C 180,E1 -21360.501,E2 -21360.501} C_VEL
LIN {X 0,Y 215.553,Z 205.536,A -85,B 0,C 180,E1 -21361.102,E2 -21361.102} C_VEL
LIN {X 0,Y 217.195,Z 159.461,A -85,B 0,C 180,E1 -21362.58,E2 -21362.58} C_VEL
LIN {X 0,Y 214.125,Z 131.067,A -85,B 0,C 180,E1 -21364.119,E2 -21364.119} C_VEL
LIN {X 0,Y 211.946,Z 124.588,A -85,B 0,C 180,E1 -21364.721,E2 -21364.721} C_VEL
LIN {X 0,Y 205.158,Z 108.577,A -85,B 0,C 180,E1 -21366.532,E2 -21366.532} C_VEL
LIN {X 0,Y 201.858,Z 101.378,A -85,B 0,C 180,E1 -21367.463,E2 -21367.463} C_VEL
LIN {X 0,Y 199.585,Z 92.623,A -85,B 0,C 180,E1 -21371.993,E2 -21371.993} C_VEL
LIN {X 0,Y 199.577,Z 92.626,A -85,B 0,C 180,E1 -21375.228,E2 -21375.228} C_VEL
LIN {X 0,Y 199.577,Z 92.624,A -85,B 0,C 180,E1 -21378.005,E2 -21378.005} C_VEL
LIN {X 0,Y 199.608,Z 92.595,A -85,B 0,C 180,E1 -21380.768,E2 -21380.768} C_VEL
LIN {X 0,Y 199.612,Z 92.619,A -85,B 0,C 180,E1 -21385.714,E2 -21385.714} C_VEL
LIN {X 0,Y 199.7,Z 92.609,A -85,B 0,C 180,E1 -21388.137,E2 -21388.137} C_VEL
LIN {X 0,Y 199.686,Z 92.602,A -85,B 0,C 180,E1 -21392.772,E2 -21392.772} C_VEL
LIN {X 0,Y 199.737,Z 92.603,A -85,B 0,C 180,E1 -21397.229,E2 -21397.229} C_VEL
LIN {X 0,Y 199.796,Z 92.592,A -85,B 0,C 180,E1 -21401.758,E2 -21401.758} C_VEL
LIN {X 0,Y 199.837,Z 92.585,A -85,B 0,C 180,E1 -21405.749,E2 -21405.749} C_VEL
LIN {X 0,Y 200.021,Z 92.563,A -85,B 0,C 180,E1 -21409.882,E2 -21409.882} C_VEL
LIN {X 0,Y 200.02,Z 92.564,A -85,B 0,C 180,E1 -21413.95,E2 -21413.95} C_VEL
LIN {X 0,Y 200.318,Z 92.523,A -85,B 0,C 180,E1 -21417.99,E2 -21417.99} C_VEL
LIN {X 0,Y 200.475,Z 92.512,A -85,B 0,C 180,E1 -21420,E2 -21420} C_VEL
LIN {X 0,Y 200.017,Z 92.552,A -85,B 0,C 180,E1 -21424.03,E2 -21424.03} C_VEL
LIN {X 0,Y 200.082,Z 92.56,A -85,B 0,C 180,E1 -21428.077,E2 -21428.077} C_VEL
LIN {X 0,Y 199.871,Z 92.572,A -85,B 0,C 180,E1 -21432.18,E2 -21432.18} C_VEL
LIN {X 0,Y 199.803,Z 92.593,A -85,B 0,C 180,E1 -21436.344,E2 -21436.344} C_VEL
LIN {X 0,Y 199.7,Z 92.594,A -85,B 0,C 180,E1 -21440.606,E2 -21440.606} C_VEL
LIN {X 0,Y 199.673,Z 92.611,A -85,B 0,C 180,E1 -21444.985,E2 -21444.985} C_VEL
LIN {X 0,Y 199.665,Z 92.613,A -85,B 0,C 180,E1 -21449.525,E2 -21449.525} C_VEL
LIN {X 0,Y 199.672,Z 92.612,A -85,B 0,C 180,E1 -21452.356,E2 -21452.356} C_VEL
LIN {X 0,Y 199.62,Z 92.622,A -85,B 0,C 180,E1 -21456.765,E2 -21456.765} C_VEL
LIN {X 0,Y 199.596,Z 92.624,A -85,B 0,C 180,E1 -21459.332,E2 -21459.332} C_VEL
LIN {X 0,Y 199.567,Z 92.625,A -85,B 0,C 180,E1 -21462.308,E2 -21462.308} C_VEL
LIN {X 0,Y 199.577,Z 92.625,A -85,B 0,C 180,E1 -21465.229,E2 -21465.229} C_VEL
LIN {X 0,Y 199.575,Z 92.623,A -85,B 0,C 180,E1 -21468.005,E2 -21468.005} C_VEL
LIN {X 0,Y 199.6,Z 92.622,A -85,B 0,C 180,E1 -21470.773,E2 -21470.773} C_VEL
LIN {X 0,Y 199.612,Z 92.62,A -85,B 0,C 180,E1 -21475.714,E2 -21475.714} C_VEL
LIN {X 0,Y 199.671,Z 92.659,A -85,B 0,C 180,E1 -21479.456,E2 -21479.456} C_VEL
LIN {X 0,Y 200.71,Z 95.537,A -85,B 0,C 180,E1 -21479.784,E2 -21479.784} C_VEL
LIN {X 0,Y 202.104,Z 97.637,A -85,B 0,C 180,E1 -21480.143,E2 -21480.143} C_VEL
LIN {X 0,Y 209.925,Z 111.734,A -85,B 0,C 180,E1 -21482.136,E2 -21482.136} C_VEL
LIN {X 0,Y 217.049,Z 126.787,A -85,B 0,C 180,E1 -21483.876,E2 -21483.876} C_VEL
LIN {X 0,Y 218.382,Z 130.593,A -85,B 0,C 180,E1 -21484.222,E2 -21484.222} C_VEL
LIN {X 0,Y 215.783,Z 193.942,A -85,B 0,C 180,E1 -21486.253,E2 -21486.253} C_VEL
LIN {X 0,Y 214.707,Z 207.437,A -85,B 0,C 180,E1 -21487.063,E2 -21487.063} C_VEL
LIN {X 0,Y 213.264,Z 220.371,A -85,B 0,C 180,E1 -21488.239,E2 -21488.239} C_VEL
LIN {X 0,Y 211.365,Z 232.891,A -85,B 0,C 180,E1 -21489.82,E2 -21489.82} C_VEL
LIN {X 0,Y 209.301,Z 244.041,A -85,B 0,C 180,E1 -21491.652,E2 -21491.652} C_VEL
LIN {X 0,Y 207.077,Z 254.104,A -85,B 0,C 180,E1 -21493.741,E2 -21493.741} C_VEL
LIN {X 0,Y 204.842,Z 263.178,A -85,B 0,C 180,E1 -21496.104,E2 -21496.104} C_VEL
LIN {X 0,Y 202.603,Z 272.016,A -85,B 0,C 180,E1 -21499.002,E2 -21499.002} C_VEL
LIN {X 0,Y 200.805,Z 279.128,A -85,B 0,C 180,E1 -21501.953,E2 -21501.953} C_VEL
LIN {X 0,Y 199.461,Z 284.798,A -85,B 0,C 180,E1 -21504.947,E2 -21504.947} C_VEL
LIN {X 0,Y 198.453,Z 289.274,A -85,B 0,C 180,E1 -21507.971,E2 -21507.971} C_VEL
LIN {X 0,Y 197.987,Z 291.638,A -85,B 0,C 180,E1 -21510.001,E2 -21510.001} C_VEL
LIN {X 0,Y 197.764,Z 293.573,A -85,B 0,C 180,E1 -21512.037,E2 -21512.037} C_VEL
LIN {X 0,Y 197.635,Z 295.792,A -85,B 0,C 180,E1 -21515.312,E2 -21515.312} C_VEL
LIN {X 0,Y 197.486,Z 296.885,A -85,B 0,C 180,E1 -21518.184,E2 -21518.184} C_VEL
LIN {X 0,Y 197.815,Z 297.129,A -85,B 0,C 180,E1 -21522.309,E2 -21522.309} C_VEL
LIN {X 0,Y 198.307,Z 296.618,A -85,B 0,C 180,E1 -21524.365,E2 -21524.365} C_VEL
LIN {X 0,Y 199.822,Z 294.406,A -85,B 0,C 180,E1 -21528.455,E2 -21528.455} C_VEL
LIN {X 0,Y 201.412,Z 291.621,A -85,B 0,C 180,E1 -21531.493,E2 -21531.493} C_VEL
LIN {X 0,Y 203.44,Z 287.791,A -85,B 0,C 180,E1 -21534.492,E2 -21534.492} C_VEL
LIN {X 0,Y 205.964,Z 282.727,A -85,B 0,C 180,E1 -21537.477,E2 -21537.477} C_VEL
LIN {X 0,Y 208.972,Z 276.496,A -85,B 0,C 180,E1 -21540.297,E2 -21540.297} C_VEL
LIN {X 0,Y 212.457,Z 268.546,A -85,B 0,C 180,E1 -21543.081,E2 -21543.081} C_VEL
LIN {X 0,Y 215.77,Z 259.903,A -85,B 0,C 180,E1 -21545.481,E2 -21545.481} C_VEL
LIN {X 0,Y 219.019,Z 250.436,A -85,B 0,C 180,E1 -21547.567,E2 -21547.567} C_VEL
LIN {X 0,Y 222.117,Z 240.583,A -85,B 0,C 180,E1 -21549.259,E2 -21549.259} C_VEL
LIN {X 0,Y 224.948,Z 229.83,A -85,B 0,C 180,E1 -21550.708,E2 -21550.708} C_VEL
LIN {X 0,Y 227.307,Z 218.202,A -85,B 0,C 180,E1 -21551.928,E2 -21551.928} C_VEL
LIN {X 0,Y 229.346,Z 205.032,A -85,B 0,C 180,E1 -21552.921,E2 -21552.921} C_VEL
LIN {X 0,Y 230.695,Z 192.109,A -85,B 0,C 180,E1 -21553.529,E2 -21553.529} C_VEL
LIN {X 0,Y 233.023,Z 146.89,A -85,B 0,C 180,E1 -21554.877,E2 -21554.877} C_VEL
LIN {X 0,Y 227.127,Z 134.198,A -85,B 0,C 180,E1 -21556.735,E2 -21556.735} C_VEL
LIN {X 0,Y 219.207,Z 121.067,A -85,B 0,C 180,E1 -21559.312,E2 -21559.312} C_VEL
LIN {X 0,Y 212.38,Z 110.833,A -85,B 0,C 180,E1 -21561.748,E2 -21561.748} C_VEL
LIN {X 0,Y 208.976,Z 106.152,A -85,B 0,C 180,E1 -21563.047,E2 -21563.047} C_VEL
LIN {X 0,Y 206.38,Z 102.43,A -85,B 0,C 180,E1 -21564.1,E2 -21564.1} C_VEL
LIN {X 0,Y 204.019,Z 99.474,A -85,B 0,C 180,E1 -21565.078,E2 -21565.078} C_VEL
LIN {X 0,Y 203.275,Z 97.965,A -85,B 0,C 180,E1 -21565.429,E2 -21565.429} C_VEL
LIN {X 0,Y 201.002,Z 95.971,A -85,B 0,C 180,E1 -21566.379,E2 -21566.379} C_VEL
LIN {X 0,Y 199.857,Z 93.629,A -85,B 0,C 180,E1 -21566.954,E2 -21566.954} C_VEL
LIN {X 0,Y 199.657,Z 92.61,A -85,B 0,C 180,E1 -21567.18,E2 -21567.18} C_VEL
LIN {X 0,Y 199.645,Z 92.603,A -85,B 0,C 180,E1 -21572.765,E2 -21572.765} C_VEL
LIN {X 0,Y 199.711,Z 92.593,A -85,B 0,C 180,E1 -21577.225,E2 -21577.225} C_VEL
LIN {X 0,Y 199.799,Z 92.582,A -85,B 0,C 180,E1 -21581.759,E2 -21581.759} C_VEL
LIN {X 0,Y 199.822,Z 92.592,A -85,B 0,C 180,E1 -21585.747,E2 -21585.747} C_VEL
LIN {X 0,Y 200.026,Z 92.563,A -85,B 0,C 180,E1 -21589.881,E2 -21589.881} C_VEL
LIN {X 0,Y 200.006,Z 92.551,A -85,B 0,C 180,E1 -21593.948,E2 -21593.948} C_VEL
LIN {X 0,Y 200.292,Z 92.528,A -85,B 0,C 180,E1 -21597.989,E2 -21597.989} C_VEL
LIN {X 0,Y 200.45,Z 92.495,A -85,B 0,C 180,E1 -21600,E2 -21600} C_VEL
LIN {X 0,Y 199.994,Z 92.566,A -85,B 0,C 180,E1 -21604.03,E2 -21604.03} C_VEL
LIN {X 0,Y 200.08,Z 92.557,A -85,B 0,C 180,E1 -21608.077,E2 -21608.077} C_VEL
LIN {X 0,Y 199.87,Z 92.568,A -85,B 0,C 180,E1 -21612.179,E2 -21612.179} C_VEL
LIN {X 0,Y 199.791,Z 92.582,A -85,B 0,C 180,E1 -21616.344,E2 -21616.344} C_VEL
LIN {X 0,Y 199.7,Z 92.604,A -85,B 0,C 180,E1 -21620.605,E2 -21620.605} C_VEL
LIN {X 0,Y 199.676,Z 92.612,A -85,B 0,C 180,E1 -21624.984,E2 -21624.984} C_VEL
LIN {X 0,Y 199.677,Z 92.611,A -85,B 0,C 180,E1 -21629.522,E2 -21629.522} C_VEL
LIN {X 0,Y 199.68,Z 92.607,A -85,B 0,C 180,E1 -21632.358,E2 -21632.358} C_VEL
LIN {X 0,Y 199.683,Z 92.59,A -85,B 0,C 180,E1 -21635.306,E2 -21635.306} C_VEL
LIN {X 0,Y 201.9,Z 99.779,A -85,B 0,C 180,E1 -21640.598,E2 -21640.598} C_VEL
LIN {X 0,Y 204.536,Z 104.191,A -85,B 0,C 180,E1 -21641.788,E2 -21641.788} C_VEL
LIN {X 0,Y 206.086,Z 106.334,A -85,B 0,C 180,E1 -21642.435,E2 -21642.435} C_VEL
LIN {X 0,Y 210.548,Z 113.577,A -85,B 0,C 180,E1 -21644.254,E2 -21644.254} C_VEL
LIN {X 0,Y 213.11,Z 117.842,A -85,B 0,C 180,E1 -21645.241,E2 -21645.241} C_VEL
LIN {X 0,Y 216.842,Z 124.396,A -85,B 0,C 180,E1 -21646.623,E2 -21646.623} C_VEL
LIN {X 0,Y 218.858,Z 129.091,A -85,B 0,C 180,E1 -21647.389,E2 -21647.389} C_VEL
LIN {X 0,Y 220.16,Z 134.427,A -85,B 0,C 180,E1 -21647.974,E2 -21647.974} C_VEL
LIN {X 0,Y 222.792,Z 149.403,A -85,B 0,C 180,E1 -21649.302,E2 -21649.302} C_VEL
LIN {X 0,Y 223.883,Z 152.903,A -85,B 0,C 180,E1 -21649.719,E2 -21649.719} C_VEL
LIN {X 0,Y 225.128,Z 156.345,A -85,B 0,C 180,E1 -21650.162,E2 -21650.162} C_VEL
LIN {X 0,Y 226.616,Z 168.102,A -85,B 0,C 180,E1 -21651,E2 -21651} C_VEL
LIN {X 0,Y 224.165,Z 210.708,A -85,B 0,C 180,E1 -21652.303,E2 -21652.303} C_VEL
LIN {X 0,Y 222.407,Z 224.341,A -85,B 0,C 180,E1 -21653.02,E2 -21653.02} C_VEL
LIN {X 0,Y 219.916,Z 237.235,A -85,B 0,C 180,E1 -21654.039,E2 -21654.039} C_VEL
LIN {X 0,Y 217.142,Z 248.147,A -85,B 0,C 180,E1 -21655.218,E2 -21655.218} C_VEL
LIN {X 0,Y 214.039,Z 258.3,A -85,B 0,C 180,E1 -21656.633,E2 -21656.633} C_VEL
LIN {X 0,Y 210.471,Z 268.845,A -85,B 0,C 180,E1 -21658.55,E2 -21658.55} C_VEL
LIN {X 0,Y 207.035,Z 277.48,A -85,B 0,C 180,E1 -21660.513,E2 -21660.513} C_VEL
LIN {X 0,Y 203.633,Z 285.451,A -85,B 0,C 180,E1 -21662.786,E2 -21662.786} C_VEL
LIN {X 0,Y 200.06,Z 293.288,A -85,B 0,C 180,E1 -21665.621,E2 -21665.621} C_VEL
LIN {X 0,Y 196.736,Z 300.486,A -85,B 0,C 180,E1 -21669.069,E2 -21669.069} C_VEL
LIN {X 0,Y 194.296,Z 305.32,A -85,B 0,C 180,E1 -21672.093,E2 -21672.093} C_VEL
LIN {X 0,Y 192.363,Z 309.052,A -85,B 0,C 180,E1 -21675.182,E2 -21675.182} C_VEL
LIN {X 0,Y 191.528,Z 310.998,A -85,B 0,C 180,E1 -21677.281,E2 -21677.281} C_VEL
LIN {X 0,Y 190.911,Z 312.517,A -85,B 0,C 180,E1 -21679.393,E2 -21679.393} C_VEL
LIN {X 0,Y 190.266,Z 314.299,A -85,B 0,C 180,E1 -21683.637,E2 -21683.637} C_VEL
LIN {X 0,Y 190.24,Z 314.629,A -85,B 0,C 180,E1 -21685.909,E2 -21685.909} C_VEL
LIN {X 0,Y 190.336,Z 314.539,A -85,B 0,C 180,E1 -21687.883,E2 -21687.883} C_VEL
LIN {X 0,Y 190.494,Z 314.026,A -85,B 0,C 180,E1 -21689.999,E2 -21689.999} C_VEL
LIN {X 0,Y 190.367,Z 313.096,A -85,B 0,C 180,E1 -21692.115,E2 -21692.115} C_VEL
LIN {X 0,Y 190.302,Z 311.689,A -85,B 0,C 180,E1 -21694.342,E2 -21694.342} C_VEL
LIN {X 0,Y 190.354,Z 308.92,A -85,B 0,C 180,E1 -21697.424,E2 -21697.424} C_VEL
LIN {X 0,Y 190.819,Z 305.033,A -85,B 0,C 180,E1 -21700.611,E2 -21700.611} C_VEL
LIN {X 0,Y 191.677,Z 299.996,A -85,B 0,C 180,E1 -21703.787,E2 -21703.787} C_VEL
LIN {X 0,Y 193.239,Z 293.678,A -85,B 0,C 180,E1 -21706.915,E2 -21706.915} C_VEL
LIN {X 0,Y 195.228,Z 285.783,A -85,B 0,C 180,E1 -21709.985,E2 -21709.985} C_VEL
LIN {X 0,Y 197.037,Z 277.629,A -85,B 0,C 180,E1 -21712.545,E2 -21712.545} C_VEL
LIN {X 0,Y 199.472,Z 267.745,A -85,B 0,C 180,E1 -21715.011,E2 -21715.011} C_VEL
LIN {X 0,Y 202.136,Z 256.732,A -85,B 0,C 180,E1 -21717.15,E2 -21717.15} C_VEL
LIN {X 0,Y 204.286,Z 245.9,A -85,B 0,C 180,E1 -21718.792,E2 -21718.792} C_VEL
LIN {X 0,Y 206.58,Z 232.865,A -85,B 0,C 180,E1 -21720.26,E2 -21720.26} C_VEL
LIN {X 0,Y 208.167,Z 220.293,A -85,B 0,C 180,E1 -21721.27,E2 -21721.27} C_VEL
LIN {X 0,Y 209.191,Z 207.094,A -85,B 0,C 180,E1 -21721.947,E2 -21721.947} C_VEL
LIN {X 0,Y 211.092,Z 161.059,A -85,B 0,C 180,E1 -21723.445,E2 -21723.445} C_VEL
LIN {X 0,Y 208.123,Z 132.83,A -85,B 0,C 180,E1 -21725.034,E2 -21725.034} C_VEL
LIN {X 0,Y 203.286,Z 120.228,A -85,B 0,C 180,E1 -21726.393,E2 -21726.393} C_VEL
LIN {X 0,Y 198.403,Z 109.11,A -85,B 0,C 180,E1 -21727.786,E2 -21727.786} C_VEL
LIN {X 0,Y 194.479,Z 100.854,A -85,B 0,C 180,E1 -21729.017,E2 -21729.017} C_VEL
LIN {X 0,Y 192.501,Z 93.507,A -85,B 0,C 180,E1 -21733.099,E2 -21733.099} C_VEL
LIN {X 0,Y 192.489,Z 93.508,A -85,B 0,C 180,E1 -21736.904,E2 -21736.904} C_VEL
LIN {X 0,Y 192.549,Z 93.472,A -85,B 0,C 180,E1 -21741.648,E2 -21741.648} C_VEL
LIN {X 0,Y 192.598,Z 93.492,A -85,B 0,C 180,E1 -21746.814,E2 -21746.814} C_VEL
LIN {X 0,Y 192.664,Z 93.482,A -85,B 0,C 180,E1 -21751.692,E2 -21751.692} C_VEL
LIN {X 0,Y 192.705,Z 93.481,A -85,B 0,C 180,E1 -21756.349,E2 -21756.349} C_VEL
LIN {X 0,Y 192.731,Z 93.47,A -85,B 0,C 180,E1 -21761.458,E2 -21761.458} C_VEL
LIN {X 0,Y 192.765,Z 93.468,A -85,B 0,C 180,E1 -21765.214,E2 -21765.214} C_VEL
LIN {X 0,Y 192.944,Z 93.443,A -85,B 0,C 180,E1 -21769.567,E2 -21769.567} C_VEL
LIN {X 0,Y 192.983,Z 93.442,A -85,B 0,C 180,E1 -21773.728,E2 -21773.728} C_VEL
LIN {X 0,Y 193.26,Z 93.401,A -85,B 0,C 180,E1 -21777.916,E2 -21777.916} C_VEL
LIN {X 0,Y 193.439,Z 93.389,A -85,B 0,C 180,E1 -21780,E2 -21780} C_VEL
LIN {X 0,Y 192.963,Z 93.429,A -85,B 0,C 180,E1 -21784.178,E2 -21784.178} C_VEL
LIN {X 0,Y 193.031,Z 93.438,A -85,B 0,C 180,E1 -21788.375,E2 -21788.375} C_VEL
LIN {X 0,Y 192.799,Z 93.45,A -85,B 0,C 180,E1 -21792.634,E2 -21792.634} C_VEL
LIN {X 0,Y 192.757,Z 93.471,A -85,B 0,C 180,E1 -21796.959,E2 -21796.959} C_VEL
LIN {X 0,Y 192.636,Z 93.471,A -85,B 0,C 180,E1 -21801.398,E2 -21801.398} C_VEL
LIN {X 0,Y 192.665,Z 93.482,A -85,B 0,C 180,E1 -21804.225,E2 -21804.225} C_VEL
LIN {X 0,Y 192.644,Z 93.488,A -85,B 0,C 180,E1 -21808.89,E2 -21808.89} C_VEL
LIN {X 0,Y 192.597,Z 93.495,A -85,B 0,C 180,E1 -21813.187,E2 -21813.187} C_VEL
LIN {X 0,Y 192.543,Z 93.499,A -85,B 0,C 180,E1 -21818.355,E2 -21818.355} C_VEL
LIN {X 0,Y 192.486,Z 93.51,A -85,B 0,C 180,E1 -21823.095,E2 -21823.095} C_VEL
LIN {X 0,Y 192.488,Z 93.506,A -85,B 0,C 180,E1 -21826.906,E2 -21826.906} C_VEL
LIN {X 0,Y 192.544,Z 93.501,A -85,B 0,C 180,E1 -21831.647,E2 -21831.647} C_VEL
LIN {X 0,Y 192.596,Z 93.488,A -85,B 0,C 180,E1 -21836.814,E2 -21836.814} C_VEL
LIN {X 0,Y 192.66,Z 93.521,A -85,B 0,C 180,E1 -21838.038,E2 -21838.038} C_VEL
LIN {X 0,Y 193.582,Z 96.251,A -85,B 0,C 180,E1 -21838.36,E2 -21838.36} C_VEL
LIN {X 0,Y 195.187,Z 98.678,A -85,B 0,C 180,E1 -21838.806,E2 -21838.806} C_VEL
LIN {X 0,Y 203.158,Z 112.671,A -85,B 0,C 180,E1 -21840.97,E2 -21840.97} C_VEL
LIN {X 0,Y 211.255,Z 129.528,A -85,B 0,C 180,E1 -21843.058,E2 -21843.058} C_VEL
LIN {X 0,Y 212.281,Z 132.904,A -85,B 0,C 180,E1 -21843.356,E2 -21843.356} C_VEL
LIN {X 0,Y 209.533,Z 194.45,A -85,B 0,C 180,E1 -21845.365,E2 -21845.365} C_VEL
LIN {X 0,Y 208.396,Z 207.918,A -85,B 0,C 180,E1 -21846.195,E2 -21846.195} C_VEL
LIN {X 0,Y 206.897,Z 220.797,A -85,B 0,C 180,E1 -21847.402,E2 -21847.402} C_VEL
LIN {X 0,Y 205.059,Z 232.509,A -85,B 0,C 180,E1 -21848.909,E2 -21848.909} C_VEL
LIN {X 0,Y 202.889,Z 243.789,A -85,B 0,C 180,E1 -21850.788,E2 -21850.788} C_VEL
LIN {X 0,Y 200.561,Z 253.978,A -85,B 0,C 180,E1 -21852.935,E2 -21852.935} C_VEL
LIN {X 0,Y 197.992,Z 263.947,A -85,B 0,C 180,E1 -21855.613,E2 -21855.613} C_VEL
LIN {X 0,Y 195.665,Z 272.71,A -85,B 0,C 180,E1 -21858.607,E2 -21858.607} C_VEL
LIN {X 0,Y 193.814,Z 279.735,A -85,B 0,C 180,E1 -21861.661,E2 -21861.661} C_VEL
LIN {X 0,Y 192.425,Z 285.339,A -85,B 0,C 180,E1 -21864.762,E2 -21864.762} C_VEL
LIN {X 0,Y 191.36,Z 289.766,A -85,B 0,C 180,E1 -21867.896,E2 -21867.896} C_VEL
LIN {X 0,Y 190.903,Z 292.105,A -85,B 0,C 180,E1 -21870.001,E2 -21870.001} C_VEL
LIN {X 0,Y 190.663,Z 294.018,A -85,B 0,C 180,E1 -21872.113,E2 -21872.113} C_VEL
LIN {X 0,Y 190.532,Z 296.007,A -85,B 0,C 180,E1 -21875.163,E2 -21875.163} C_VEL
LIN {X 0,Y 190.412,Z 297.241,A -85,B 0,C 180,E1 -21878.491,E2 -21878.491} C_VEL
LIN {X 0,Y 190.508,Z 297.536,A -85,B 0,C 180,E1 -21880.63,E2 -21880.63} C_VEL
LIN {X 0,Y 190.802,Z 297.428,A -85,B 0,C 180,E1 -21882.769,E2 -21882.769} C_VEL
LIN {X 0,Y 192.077,Z 295.956,A -85,B 0,C 180,E1 -21887.021,E2 -21887.021} C_VEL
LIN {X 0,Y 192.998,Z 294.629,A -85,B 0,C 180,E1 -21889.132,E2 -21889.132} C_VEL
LIN {X 0,Y 194.7,Z 291.797,A -85,B 0,C 180,E1 -21892.273,E2 -21892.273} C_VEL
LIN {X 0,Y 196.901,Z 287.916,A -85,B 0,C 180,E1 -21895.361,E2 -21895.361} C_VEL
LIN {X 0,Y 199.787,Z 282.462,A -85,B 0,C 180,E1 -21898.603,E2 -21898.603} C_VEL
LIN {X 0,Y 203.341,Z 275.249,A -85,B 0,C 180,E1 -21901.809,E2 -21901.809} C_VEL
LIN {X 0,Y 207.108,Z 266.964,A -85,B 0,C 180,E1 -21904.639,E2 -21904.639} C_VEL
LIN {X 0,Y 210.419,Z 258.416,A -85,B 0,C 180,E1 -21906.957,E2 -21906.957} C_VEL
LIN {X 0,Y 213.772,Z 248.989,A -85,B 0,C 180,E1 -21908.959,E2 -21908.959} C_VEL
LIN {X 0,Y 217.413,Z 237.247,A -85,B 0,C 180,E1 -21910.89,E2 -21910.89} C_VEL
LIN {X 0,Y 220.264,Z 226.297,A -85,B 0,C 180,E1 -21912.26,E2 -21912.26} C_VEL
LIN {X 0,Y 222.413,Z 214.869,A -85,B 0,C 180,E1 -21913.382,E2 -21913.382} C_VEL
LIN {X 0,Y 224.392,Z 201.592,A -85,B 0,C 180,E1 -21914.264,E2 -21914.264} C_VEL
LIN {X 0,Y 225.486,Z 189.063,A -85,B 0,C 180,E1 -21914.8,E2 -21914.8} C_VEL
LIN {X 0,Y 227.617,Z 149.151,A -85,B 0,C 180,E1 -21915.989,E2 -21915.989} C_VEL
LIN {X 0,Y 222.365,Z 137.96,A -85,B 0,C 180,E1 -21917.73,E2 -21917.73} C_VEL
LIN {X 0,Y 215.06,Z 125.63,A -85,B 0,C 180,E1 -21920.241,E2 -21920.241} C_VEL
LIN {X 0,Y 208.508,Z 115.741,A -85,B 0,C 180,E1 -21922.699,E2 -21922.699} C_VEL
LIN {X 0,Y 205.473,Z 111.517,A -85,B 0,C 180,E1 -21923.917,E2 -21923.917} C_VEL
LIN {X 0,Y 202.816,Z 107.809,A -85,B 0,C 180,E1 -21925.04,E2 -21925.04} C_VEL
LIN {X 0,Y 200.323,Z 104.239,A -85,B 0,C 180,E1 -21926.154,E2 -21926.154} C_VEL
LIN {X 0,Y 197.416,Z 100.912,A -85,B 0,C 180,E1 -21927.478,E2 -21927.478} C_VEL
LIN {X 0,Y 196.185,Z 98.755,A -85,B 0,C 180,E1 -21928.111,E2 -21928.111} C_VEL
LIN {X 0,Y 193.898,Z 96.785,A -85,B 0,C 180,E1 -21929.204,E2 -21929.204} C_VEL
LIN {X 0,Y 192.802,Z 94.567,A -85,B 0,C 180,E1 -21929.832,E2 -21929.832} C_VEL
LIN {X 0,Y 192.562,Z 93.496,A -85,B 0,C 180,E1 -21930.049,E2 -21930.049} C_VEL
LIN {X 0,Y 192.571,Z 93.491,A -85,B 0,C 180,E1 -21934.026,E2 -21934.026} C_VEL
LIN {X 0,Y 192.682,Z 93.472,A -85,B 0,C 180,E1 -21936.345,E2 -21936.345} C_VEL
LIN {X 0,Y 192.734,Z 93.463,A -85,B 0,C 180,E1 -21941.459,E2 -21941.459} C_VEL
LIN {X 0,Y 192.752,Z 93.476,A -85,B 0,C 180,E1 -21945.212,E2 -21945.212} C_VEL
LIN {X 0,Y 192.949,Z 93.44,A -85,B 0,C 180,E1 -21949.566,E2 -21949.566} C_VEL
LIN {X 0,Y 192.97,Z 93.427,A -85,B 0,C 180,E1 -21953.727,E2 -21953.727} C_VEL
LIN {X 0,Y 193.236,Z 93.407,A -85,B 0,C 180,E1 -21957.915,E2 -21957.915} C_VEL
LIN {X 0,Y 193.417,Z 93.371,A -85,B 0,C 180,E1 -21960,E2 -21960} C_VEL
LIN {X 0,Y 192.941,Z 93.441,A -85,B 0,C 180,E1 -21964.177,E2 -21964.177} C_VEL
LIN {X 0,Y 193.03,Z 93.437,A -85,B 0,C 180,E1 -21968.374,E2 -21968.374} C_VEL
LIN {X 0,Y 192.797,Z 93.451,A -85,B 0,C 180,E1 -21972.633,E2 -21972.633} C_VEL
LIN {X 0,Y 192.75,Z 93.456,A -85,B 0,C 180,E1 -21976.959,E2 -21976.959} C_VEL
LIN {X 0,Y 192.637,Z 93.476,A -85,B 0,C 180,E1 -21981.397,E2 -21981.397} C_VEL
LIN {X 0,Y 192.667,Z 93.483,A -85,B 0,C 180,E1 -21984.224,E2 -21984.224} C_VEL
LIN {X 0,Y 192.653,Z 93.488,A -85,B 0,C 180,E1 -21988.891,E2 -21988.891} C_VEL
LIN {X 0,Y 192.613,Z 93.514,A -85,B 0,C 180,E1 -21992.941,E2 -21992.941} C_VEL
LIN {X 0,Y 194.43,Z 99.204,A -85,B 0,C 180,E1 -21997.605,E2 -21997.605} C_VEL
LIN {X 0,Y 196.925,Z 103.291,A -85,B 0,C 180,E1 -21998.895,E2 -21998.895} C_VEL
LIN {X 0,Y 198.907,Z 105.862,A -85,B 0,C 180,E1 -21999.828,E2 -21999.828} C_VEL
LIN {X 0,Y 201.83,Z 110.425,A -85,B 0,C 180,E1 -22001.177,E2 -22001.177} C_VEL
LIN {X 0,Y 206.595,Z 118.214,A -85,B 0,C 180,E1 -22003.237,E2 -22003.237} C_VEL
LIN {X 0,Y 209.674,Z 123.497,A -85,B 0,C 180,E1 -22004.487,E2 -22004.487} C_VEL
LIN {X 0,Y 215.825,Z 134.887,A -85,B 0,C 180,E1 -22006.836,E2 -22006.836} C_VEL
LIN {X 0,Y 222.106,Z 148.587,A -85,B 0,C 180,E1 -22009.098,E2 -22009.098} C_VEL
LIN {X 0,Y 223.883,Z 152.903,A -85,B 0,C 180,E1 -22009.719,E2 -22009.719} C_VEL
LIN {X 0,Y 224.7,Z 156.431,A -85,B 0,C 180,E1 -22010.064,E2 -22010.064} C_VEL
LIN {X 0,Y 224.687,Z 162.226,A -85,B 0,C 180,E1 -22010.309,E2 -22010.309} C_VEL
LIN {X 0,Y 223.722,Z 168.123,A -85,B 0,C 180,E1 -22010.334,E2 -22010.334} C_VEL
LIN {X 0,Y 220.981,Z 180.413,A -85,B 0,C 180,E1 -22010.214,E2 -22010.214} C_VEL
LIN {X 0,Y 220.488,Z 184.555,A -85,B 0,C 180,E1 -22010.276,E2 -22010.276} C_VEL
LIN {X 0,Y 218.801,Z 210.789,A -85,B 0,C 180,E1 -22011.103,E2 -22011.103} C_VEL
LIN {X 0,Y 216.946,Z 224.475,A -85,B 0,C 180,E1 -22011.838,E2 -22011.838} C_VEL
LIN {X 0,Y 214.472,Z 236.808,A -85,B 0,C 180,E1 -22012.83,E2 -22012.83} C_VEL
LIN {X 0,Y 211.367,Z 248.531,A -85,B 0,C 180,E1 -22014.123,E2 -22014.123} C_VEL
LIN {X 0,Y 208.165,Z 258.554,A -85,B 0,C 180,E1 -22015.562,E2 -22015.562} C_VEL
LIN {X 0,Y 204.451,Z 269,A -85,B 0,C 180,E1 -22017.512,E2 -22017.512} C_VEL
LIN {X 0,Y 200.897,Z 277.556,A -85,B 0,C 180,E1 -22019.518,E2 -22019.518} C_VEL
LIN {X 0,Y 197.329,Z 285.461,A -85,B 0,C 180,E1 -22021.841,E2 -22021.841} C_VEL
LIN {X 0,Y 193.598,Z 293.215,A -85,B 0,C 180,E1 -22024.751,E2 -22024.751} C_VEL
LIN {X 0,Y 190.112,Z 300.366,A -85,B 0,C 180,E1 -22028.304,E2 -22028.304} C_VEL
LIN {X 0,Y 187.534,Z 305.157,A -85,B 0,C 180,E1 -22031.424,E2 -22031.424} C_VEL
LIN {X 0,Y 185.478,Z 308.847,A -85,B 0,C 180,E1 -22034.618,E2 -22034.618} C_VEL
LIN {X 0,Y 184.575,Z 310.774,A -85,B 0,C 180,E1 -22036.793,E2 -22036.793} C_VEL
LIN {X 0,Y 183.9,Z 312.257,A -85,B 0,C 180,E1 -22038.983,E2 -22038.983} C_VEL
LIN {X 0,Y 183.197,Z 314.003,A -85,B 0,C 180,E1 -22043.391,E2 -22043.391} C_VEL
LIN {X 0,Y 183.147,Z 314.311,A -85,B 0,C 180,E1 -22046.12,E2 -22046.12} C_VEL
LIN {X 0,Y 183.408,Z 313.662,A -85,B 0,C 180,E1 -22049.999,E2 -22049.999} C_VEL
LIN {X 0,Y 183.267,Z 312.714,A -85,B 0,C 180,E1 -22052.197,E2 -22052.197} C_VEL
LIN {X 0,Y 183.227,Z 311.363,A -85,B 0,C 180,E1 -22054.399,E2 -22054.399} C_VEL
LIN {X 0,Y 183.304,Z 308.482,A -85,B 0,C 180,E1 -22057.711,E2 -22057.711} C_VEL
LIN {X 0,Y 183.808,Z 304.554,A -85,B 0,C 180,E1 -22061.021,E2 -22061.021} C_VEL
LIN {X 0,Y 184.754,Z 299.475,A -85,B 0,C 180,E1 -22064.315,E2 -22064.315} C_VEL
LIN {X 0,Y 186.391,Z 293.099,A -85,B 0,C 180,E1 -22067.556,E2 -22067.556} C_VEL
LIN {X 0,Y 188.409,Z 285.501,A -85,B 0,C 180,E1 -22070.6,E2 -22070.6} C_VEL
LIN {X 0,Y 190.421,Z 276.905,A -85,B 0,C 180,E1 -22073.375,E2 -22073.375} C_VEL
LIN {X 0,Y 192.744,Z 268.026,A -85,B 0,C 180,E1 -22075.657,E2 -22075.657} C_VEL
LIN {X 0,Y 195.503,Z 257.175,A -85,B 0,C 180,E1 -22077.86,E2 -22077.86} C_VEL
LIN {X 0,Y 197.722,Z 246.569,A -85,B 0,C 180,E1 -22079.55,E2 -22079.55} C_VEL
LIN {X 0,Y 200.083,Z 233.806,A -85,B 0,C 180,E1 -22081.057,E2 -22081.057} C_VEL
LIN {X 0,Y 201.835,Z 221.005,A -85,B 0,C 180,E1 -22082.147,E2 -22082.147} C_VEL
LIN {X 0,Y 202.93,Z 208.631,A -85,B 0,C 180,E1 -22082.834,E2 -22082.834} C_VEL
LIN {X 0,Y 204.877,Z 160.716,A -85,B 0,C 180,E1 -22084.467,E2 -22084.467} C_VEL
LIN {X 0,Y 202.225,Z 134.798,A -85,B 0,C 180,E1 -22085.984,E2 -22085.984} C_VEL
LIN {X 0,Y 195.21,Z 117.195,A -85,B 0,C 180,E1 -22088.072,E2 -22088.072} C_VEL
LIN {X 0,Y 189.208,Z 104.781,A -85,B 0,C 180,E1 -22089.906,E2 -22089.906} C_VEL
LIN {X 0,Y 187.119,Z 100.52,A -85,B 0,C 180,E1 -22090.629,E2 -22090.629} C_VEL
LIN {X 0,Y 185.441,Z 94.386,A -85,B 0,C 180,E1 -22094.231,E2 -22094.231} C_VEL
LIN {X 0,Y 185.468,Z 94.367,A -85,B 0,C 180,E1 -22099.275,E2 -22099.275} C_VEL
LIN {X 0,Y 185.504,Z 94.355,A -85,B 0,C 180,E1 -22102.711,E2 -22102.711} C_VEL
LIN {X 0,Y 185.545,Z 94.372,A -85,B 0,C 180,E1 -22107.976,E2 -22107.976} C_VEL
LIN {X 0,Y 185.581,Z 94.369,A -85,B 0,C 180,E1 -22110.576,E2 -22110.576} C_VEL
LIN {X 0,Y 185.587,Z 94.366,A -85,B 0,C 180,E1 -22115.383,E2 -22115.383} C_VEL
LIN {X 0,Y 185.674,Z 94.345,A -85,B 0,C 180,E1 -22121.133,E2 -22121.133} C_VEL
LIN {X 0,Y 185.696,Z 94.351,A -85,B 0,C 180,E1 -22124.638,E2 -22124.638} C_VEL
LIN {X 0,Y 185.887,Z 94.32,A -85,B 0,C 180,E1 -22129.418,E2 -22129.418} C_VEL
LIN {X 0,Y 185.946,Z 94.32,A -85,B 0,C 180,E1 -22133.49,E2 -22133.49} C_VEL
LIN {X 0,Y 186.204,Z 94.279,A -85,B 0,C 180,E1 -22137.837,E2 -22137.837} C_VEL
LIN {X 0,Y 186.403,Z 94.265,A -85,B 0,C 180,E1 -22140,E2 -22140} C_VEL
LIN {X 0,Y 185.909,Z 94.306,A -85,B 0,C 180,E1 -22144.337,E2 -22144.337} C_VEL
LIN {X 0,Y 185.979,Z 94.315,A -85,B 0,C 180,E1 -22148.695,E2 -22148.695} C_VEL
LIN {X 0,Y 185.726,Z 94.329,A -85,B 0,C 180,E1 -22153.124,E2 -22153.124} C_VEL
LIN {X 0,Y 185.69,Z 94.352,A -85,B 0,C 180,E1 -22157.626,E2 -22157.626} C_VEL
LIN {X 0,Y 185.597,Z 94.349,A -85,B 0,C 180,E1 -22162.252,E2 -22162.252} C_VEL
LIN {X 0,Y 185.561,Z 94.367,A -85,B 0,C 180,E1 -22167.033,E2 -22167.033} C_VEL
LIN {X 0,Y 185.578,Z 94.368,A -85,B 0,C 180,E1 -22169.494,E2 -22169.494} C_VEL
LIN {X 0,Y 185.498,Z 94.376,A -85,B 0,C 180,E1 -22174.633,E2 -22174.633} C_VEL
LIN {X 0,Y 185.501,Z 94.377,A -85,B 0,C 180,E1 -22177.315,E2 -22177.315} C_VEL
LIN {X 0,Y 185.462,Z 94.383,A -85,B 0,C 180,E1 -22180.722,E2 -22180.722} C_VEL
LIN {X 0,Y 185.458,Z 94.385,A -85,B 0,C 180,E1 -22186.056,E2 -22186.056} C_VEL
LIN {X 0,Y 185.46,Z 94.382,A -85,B 0,C 180,E1 -22189.894,E2 -22189.894} C_VEL
LIN {X 0,Y 185.502,Z 94.378,A -85,B 0,C 180,E1 -22192.715,E2 -22192.715} C_VEL
LIN {X 0,Y 185.521,Z 94.37,A -85,B 0,C 180,E1 -22196.452,E2 -22196.452} C_VEL
LIN {X 0,Y 186.649,Z 97.36,A -85,B 0,C 180,E1 -22196.862,E2 -22196.862} C_VEL
LIN {X 0,Y 188.155,Z 99.392,A -85,B 0,C 180,E1 -22197.306,E2 -22197.306} C_VEL
LIN {X 0,Y 197.08,Z 114.853,A -85,B 0,C 180,E1 -22199.899,E2 -22199.899} C_VEL
LIN {X 0,Y 205.115,Z 131.516,A -85,B 0,C 180,E1 -22202.095,E2 -22202.095} C_VEL
LIN {X 0,Y 206.151,Z 134.401,A -85,B 0,C 180,E1 -22202.392,E2 -22202.392} C_VEL
LIN {X 0,Y 203.352,Z 194.766,A -85,B 0,C 180,E1 -22204.414,E2 -22204.414} C_VEL
LIN {X 0,Y 202.17,Z 208.044,A -85,B 0,C 180,E1 -22205.247,E2 -22205.247} C_VEL
LIN {X 0,Y 200.7,Z 220.158,A -85,B 0,C 180,E1 -22206.39,E2 -22206.39} C_VEL
LIN {X 0,Y 198.807,Z 232.114,A -85,B 0,C 180,E1 -22207.939,E2 -22207.939} C_VEL
LIN {X 0,Y 196.508,Z 243.529,A -85,B 0,C 180,E1 -22209.866,E2 -22209.866} C_VEL
LIN {X 0,Y 194.084,Z 253.824,A -85,B 0,C 180,E1 -22212.074,E2 -22212.074} C_VEL
LIN {X 0,Y 191.589,Z 263.094,A -85,B 0,C 180,E1 -22214.577,E2 -22214.577} C_VEL
LIN {X 0,Y 189.129,Z 272.051,A -85,B 0,C 180,E1 -22217.663,E2 -22217.663} C_VEL
LIN {X 0,Y 187.069,Z 279.279,A -85,B 0,C 180,E1 -22220.813,E2 -22220.813} C_VEL
LIN {X 0,Y 185.823,Z 284.16,A -85,B 0,C 180,E1 -22223.486,E2 -22223.486} C_VEL
LIN {X 0,Y 184.618,Z 288.915,A -85,B 0,C 180,E1 -22226.727,E2 -22226.727} C_VEL
LIN {X 0,Y 183.819,Z 292.571,A -85,B 0,C 180,E1 -22230.001,E2 -22230.001} C_VEL
LIN {X 0,Y 183.566,Z 294.462,A -85,B 0,C 180,E1 -22232.195,E2 -22232.195} C_VEL
LIN {X 0,Y 183.46,Z 296.275,A -85,B 0,C 180,E1 -22235.111,E2 -22235.111} C_VEL
LIN {X 0,Y 183.331,Z 297.597,A -85,B 0,C 180,E1 -22238.821,E2 -22238.821} C_VEL
LIN {X 0,Y 183.451,Z 297.871,A -85,B 0,C 180,E1 -22241.044,E2 -22241.044} C_VEL
LIN {X 0,Y 183.801,Z 297.719,A -85,B 0,C 180,E1 -22243.264,E2 -22243.264} C_VEL
LIN {X 0,Y 185.219,Z 296.202,A -85,B 0,C 180,E1 -22247.672,E2 -22247.672} C_VEL
LIN {X 0,Y 186.194,Z 294.852,A -85,B 0,C 180,E1 -22249.86,E2 -22249.86} C_VEL
LIN {X 0,Y 188.042,Z 291.975,A -85,B 0,C 180,E1 -22253.107,E2 -22253.107} C_VEL
LIN {X 0,Y 190.412,Z 288.044,A -85,B 0,C 180,E1 -22256.291,E2 -22256.291} C_VEL
LIN {X 0,Y 193.781,Z 281.939,A -85,B 0,C 180,E1 -22259.914,E2 -22259.914} C_VEL
LIN {X 0,Y 197.265,Z 275.233,A -85,B 0,C 180,E1 -22262.91,E2 -22262.91} C_VEL
LIN {X 0,Y 201.237,Z 266.87,A -85,B 0,C 180,E1 -22265.802,E2 -22265.802} C_VEL
LIN {X 0,Y 204.685,Z 258.2,A -85,B 0,C 180,E1 -22268.174,E2 -22268.174} C_VEL
